KUKA KRL program: MyProgram_098().src

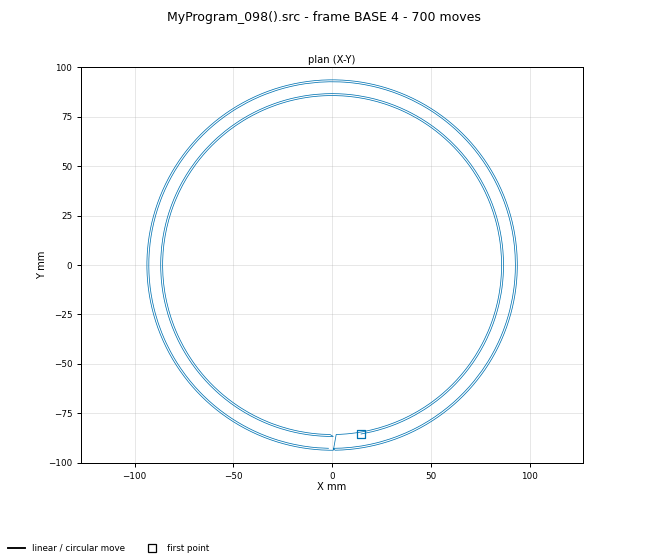
[picture p0: tool path of MyProgram_098().src in frame BASE 4, 700 of 700 moves have a stored position in this frame; points joined in program order, loops and branches not executed]
&ACCESS RVP
&REL 1
&PARAM TEMPLATE = C:\KRC\Roboter\Template\vorgabe
&PARAM EDITMASK = *
DEF MyProgram_098()
; ---- Setting reference (Base) ----
$BASE = BASE_DATA[4]

; --------------------------
; ---- Setting tool (TCP) ----
$TOOL = TOOL_DATA[3]
; --------------------------

$VEL.CP = VEL_APROX_PRINT
Startdeposition()
$VEL.CP = VEL_PRINT
LIN {X 14.6737,Y -85.5228,Z 90,A -84.3655,B 24.9258,C -1.989,E1 25.029,E2 169.2981} C_DIS
LIN {X 20.2856,Y -84.3677,Z 90,A -80.6832,B 24.9258,C -1.989,E1 25.0391,E2 165.6204} C_DIS
LIN {X 23.2527,Y -83.5992,Z 90,A -78.5972,B 24.9255,C -1.9933,E1 25.0447,E2 163.5279} C_DIS
LIN {X 26.6755,Y -82.5697,Z 90,A -75.7569,B 24.9241,C -2.0121,E1 25.0524,E2 160.6482} C_DIS
LIN {X 29.8401,Y -81.4795,Z 90,A -74.198,B 24.9255,C -1.9932,E1 25.0564,E2 159.1372} C_DIS
LIN {X 32.722,Y -80.3655,Z 90,A -72.0573,B 24.925,C -1.9994,E1 25.0619,E2 156.9867} C_DIS
LIN {X 35.8348,Y -79.0269,Z 90,A -69.6084,B 24.9243,C -2.0099,E1 25.0682,E2 154.5189} C_DIS
LIN {X 39.2577,Y -77.3837,Z 90,A -67.354,B 24.9246,C -2.0054,E1 25.0738,E2 152.2811} C_DIS
LIN {X 42.0598,Y -75.8972,Z 90,A -65.2291,B 24.9242,C -2.0101,E1 25.0791,E2 150.1513} C_DIS
LIN {X 46.6646,Y -73.1561,Z 90,A -62.0519,B 24.9247,C -2.0044,E1 25.0866,E2 146.9974} C_DIS
LIN {X 49.1042,Y -71.5429,Z 90,A -59.5239,B 24.9228,C -2.0285,E1 25.0926,E2 144.421} C_DIS
LIN {X 52.849,Y -68.8211,Z 90,A -56.8631,B 24.9234,C -2.0213,E1 25.0985,E2 141.7866} C_DIS
LIN {X 55.1312,Y -67.0079,Z 90,A -54.4863,B 24.9219,C -2.0411,E1 25.1037,E2 139.3722} C_DIS
LIN {X 57.7938,Y -64.7243,Z 90,A -52.5166,B 24.9224,C -2.0344,E1 25.1078,E2 137.426} C_DIS
LIN {X 60.5413,Y -62.1634,Z 90,A -50.2244,B 24.9224,C -2.0338,E1 25.1124,E2 135.1446} C_DIS
LIN {X 62.5386,Y -60.1521,Z 90,A -47.6066,B 24.9201,C -2.0643,E1 25.1176,E2 132.4661} C_DIS
LIN {X 64.9854,Y -57.5021,Z 90,A -45.8844,B 24.9214,C -2.0474,E1 25.1207,E2 130.7915} C_DIS
LIN {X 67.2469,Y -54.8385,Z 90,A -43.5543,B 24.9209,C -2.0542,E1 25.1249,E2 128.456} C_DIS
LIN {X 69.1339,Y -52.4405,Z 90,A -41.4737,B 24.9203,C -2.0619,E1 25.1285,E2 126.3672} C_DIS
LIN {X 71.5187,Y -49.139,Z 90,A -38.7198,B 24.9195,C -2.0715,E1 25.1329,E2 123.6039} C_DIS
LIN {X 73.5355,Y -46.0638,Z 90,A -35.8783,B 24.9179,C -2.0929,E1 25.1372,E2 120.7264} C_DIS
LIN {X 75.3159,Y -43.0915,Z 90,A -34.2647,B 24.9192,C -2.0758,E1 25.1394,E2 119.1613} C_DIS
LIN {X 76.7944,Y -40.3975,Z 90,A -32.1566,B 24.9185,C -2.0845,E1 25.1422,E2 117.0438} C_DIS
LIN {X 78.2764,Y -37.4454,Z 90,A -30.0963,B 24.9183,C -2.0868,E1 25.1447,E2 114.9892} C_DIS
LIN {X 80.2361,Y -33.0399,Z 90,A -26.7347,B 24.9171,C -2.1026,E1 25.1485,E2 111.6085} C_DIS
LIN {X 81.5916,Y -29.5328,Z 90,A -24.3204,B 24.9167,C -2.1079,E1 25.1508,E2 109.1953} C_DIS
LIN {X 82.6553,Y -26.4109,Z 90,A -22.0449,B 24.9159,C -2.1181,E1 25.1528,E2 106.9086} C_DIS
LIN {X 83.6832,Y -22.947,Z 90,A -19.8263,B 24.9157,C -2.1197,E1 25.1545,E2 104.6989} C_DIS
LIN {X 84.5153,Y -19.6601,Z 90,A -17.6432,B 24.9153,C -2.1248,E1 25.156,E2 102.5163} C_DIS
LIN {X 85.6245,Y -14.0659,Z 90,A -14.0298,B 24.9148,C -2.1314,E1 25.1579,E2 98.9085} C_DIS
LIN {X 86.0338,Y -11.2937,Z 90,A -12.3098,B 24.9147,C -2.1328,E1 25.1585,E2 97.1954} C_DIS
LIN {X 86.3255,Y -8.7923,Z 90,A -10.324,B 24.9133,C -2.1494,E1 25.1591,E2 95.182} C_DIS
LIN {X 86.6108,Y -5.3073,Z 90,A -7.9931,B 24.9127,C -2.1576,E1 25.1596,E2 92.8457} C_DIS
LIN {X 86.7486,Y -2.0565,Z 90,A -6.0028,B 24.9126,C -2.1589,E1 25.1598,E2 90.8641} C_DIS
LIN {X 86.7724,Y 0.3329,Z 90,A -4.3418,B 24.9119,C -2.1669,E1 25.1598,E2 89.1941} C_DIS
LIN {X 86.6858,Y 3.8646,Z 90,A -2.0074,B 24.9113,C -2.1744,E1 25.1595,E2 86.8558} C_DIS
LIN {X 86.4689,Y 7.2509,Z 90,A 0.1968,B 24.9108,C -2.1802,E1 25.1591,E2 84.651} C_DIS
LIN {X 86.1374,Y 10.4803,Z 90,A 2.3644,B 24.9102,C -2.1879,E1 25.1584,E2 82.4782} C_DIS
LIN {X 85.6296,Y 14.0351,Z 90,A 4.6778,B 24.9098,C -2.1933,E1 25.1574,E2 80.1656} C_DIS
LIN {X 85.1173,Y 16.8701,Z 90,A 6.6048,B 24.9092,C -2.2,E1 25.1564,E2 78.234} C_DIS
LIN {X 84.3903,Y 20.1931,Z 90,A 9.1136,B 24.9079,C -2.2161,E1 25.1548,E2 75.7017} C_DIS
LIN {X 83.2328,Y 24.5287,Z 90,A 11.6474,B 24.9084,C -2.2101,E1 25.1529,E2 73.1967} C_DIS
LIN {X 82.1608,Y 27.9101,Z 90,A 14.0041,B 24.9078,C -2.2176,E1 25.1509,E2 70.8357} C_DIS
LIN {X 81.0713,Y 30.9326,Z 90,A 16.1391,B 24.9072,C -2.2242,E1 25.1488,E2 68.6968} C_DIS
LIN {X 79.8847,Y 33.8794,Z 90,A 18.3025,B 24.9065,C -2.2326,E1 25.1465,E2 66.5256} C_DIS
LIN {X 78.4299,Y 37.1259,Z 90,A 20.3817,B 24.9067,C -2.2298,E1 25.1441,E2 64.4642} C_DIS
LIN {X 77.2493,Y 39.5206,Z 90,A 22.2334,B 24.9061,C -2.2378,E1 25.1417,E2 62.6036} C_DIS
LIN {X 75.2931,Y 43.1312,Z 90,A 24.6796,B 24.9062,C -2.236,E1 25.1385,E2 60.1744} C_DIS
LIN {X 74.1236,Y 45.1114,Z 90,A 26.4463,B 24.9052,C -2.2485,E1 25.1359,E2 58.3871} C_DIS
LIN {X 72.4967,Y 47.6821,Z 90,A 28.5137,B 24.9045,C -2.2557,E1 25.1328,E2 56.3132} C_DIS
LIN {X 70.2728,Y 50.9045,Z 90,A 31.1629,B 24.9038,C -2.2643,E1 25.1285,E2 53.6565} C_DIS
LIN {X 67.8225,Y 54.1259,Z 90,A 33.8258,B 24.9033,C -2.2704,E1 25.1239,E2 50.9918} C_DIS
LIN {X 65.5568,Y 56.8483,Z 90,A 36.1165,B 24.903,C -2.2742,E1 25.1198,E2 48.7027} C_DIS
LIN {X 63.2083,Y 59.4478,Z 90,A 38.8418,B 24.9013,C -2.2933,E1 25.1145,E2 45.9441} C_DIS
LIN {X 59.9076,Y 62.7742,Z 90,A 42.5078,B 24.8991,C -2.3192,E1 25.1071,E2 42.232} C_DIS
LIN {X 56.1883,Y 66.1228,Z 90,A 44.5817,B 24.9021,C -2.284,E1 25.1029,E2 40.2496} C_DIS
LIN {X 53.9722,Y 67.944,Z 90,A 46.6317,B 24.9014,C -2.2927,E1 25.0984,E2 38.1867} C_DIS
LIN {X 51.2627,Y 70.0105,Z 90,A 49.0796,B 24.9005,C -2.3032,E1 25.0929,E2 35.7226} C_DIS
LIN {X 48.4048,Y 72.0167,Z 90,A 51.2483,B 24.9005,C -2.3024,E1 25.0879,E2 33.5631} C_DIS
LIN {X 45.433,Y 73.9281,Z 90,A 53.5185,B 24.9005,C -2.3039,E1 25.0825,E2 31.2967} C_DIS
LIN {X 42.7507,Y 75.5114,Z 90,A 55.582,B 24.9001,C -2.3071,E1 25.0776,E2 29.232} C_DIS
LIN {X 40.0108,Y 76.9981,Z 90,A 57.4695,B 24.9004,C -2.3042,E1 25.0729,E2 27.3566} C_DIS
LIN {X 38.1158,Y 77.9535,Z 90,A 59.4503,B 24.8986,C -2.325,E1 25.0679,E2 25.3319} C_DIS
LIN {X 34.568,Y 79.5889,Z 90,A 61.647,B 24.8994,C -2.3153,E1 25.0623,E2 23.1635} C_DIS
LIN {X 31.3475,Y 80.9125,Z 90,A 63.8972,B 24.8994,C -2.316,E1 25.0565,E2 20.9168} C_DIS
LIN {X 28.2615,Y 82.0419,Z 90,A 66.0927,B 24.8991,C -2.3187,E1 25.0507,E2 18.7192} C_DIS
LIN {X 25.1389,Y 83.0518,Z 90,A 68.3337,B 24.8988,C -2.3228,E1 25.0447,E2 16.4727} C_DIS
LIN {X 21.4921,Y 84.0681,Z 90,A 70.6005,B 24.8993,C -2.3169,E1 25.0386,E2 14.2234} C_DIS
LIN {X 18.0347,Y 84.8782,Z 90,A 73.1039,B 24.8987,C -2.3231,E1 25.0318,E2 11.7086} C_DIS
LIN {X 12.9971,Y 85.7932,Z 90,A 76.2246,B 24.8994,C -2.316,E1 25.0233,E2 8.608} C_DIS
LIN {X 10.3284,Y 86.1552,Z 90,A 78.166,B 24.8989,C -2.3216,E1 25.0179,E2 6.655} C_DIS
LIN {X 7.047,Y 86.4852,Z 90,A 80.4053,B 24.8987,C -2.3237,E1 25.0116,E2 4.4119} C_DIS
LIN {X 3.4616,Y 86.7031,Z 90,A 82.8215,B 24.8986,C -2.325,E1 25.0049,E2 1.9934} C_DIS
LIN {X -0.1215,Y 86.7726,Z 90,A 85.1767,B 24.8986,C -2.3243,E1 24.9983,E2 -0.3598} C_DIS
LIN {X -3.486,Y 86.702,Z 90,A 88.3102,B 24.8962,C -2.3522,E1 24.9894,E2 -3.5602} C_DIS
LIN {X -8.2682,Y 86.3774,Z 90,A 90.3011,B 24.8995,C -2.3141,E1 24.9841,E2 -5.4615} C_DIS
LIN {X -10.9104,Y 86.0834,Z 90,A 92.2875,B 24.899,C -2.3202,E1 24.9785,E2 -7.4637} C_DIS
LIN {X -14.2435,Y 85.5948,Z 90,A 94.3609,B 24.8995,C -2.314,E1 24.9728,E2 -9.5243} C_DIS
LIN {X -18.3888,Y 84.8009,Z 90,A 97.2041,B 24.8995,C -2.3135,E1 24.9651,E2 -12.3694} C_DIS
LIN {X -20.776,Y 84.2481,Z 90,A 98.7974,B 24.8998,C -2.3112,E1 24.9607,E2 -13.9594} C_DIS
LIN {X -23.5949,Y 83.5022,Z 90,A 100.7155,B 24.9,C -2.309,E1 24.9556,E2 -15.8753} C_DIS
LIN {X -26.4229,Y 82.6514,Z 90,A 102.7582,B 24.9,C -2.3096,E1 24.9501,E2 -17.9229} C_DIS
LIN {X -29.1641,Y 81.7252,Z 90,A 104.6404,B 24.9002,C -2.3063,E1 24.9452,E2 -19.8011} C_DIS
LIN {X -32.9874,Y 80.2574,Z 90,A 106.9907,B 24.9014,C -2.2921,E1 24.9391,E2 -22.1227} C_DIS
LIN {X -36.8189,Y 78.5732,Z 90,A 110.1387,B 24.9008,C -2.2995,E1 24.931,E2 -25.2958} C_DIS
LIN {X -39.6003,Y 77.2086,Z 90,A 112.1958,B 24.901,C -2.2965,E1 24.9259,E2 -27.3513} C_DIS
LIN {X -42.1651,Y 75.8384,Z 90,A 114.2188,B 24.901,C -2.2963,E1 24.9209,E2 -29.3795} C_DIS
LIN {X -45.1483,Y 74.1011,Z 90,A 116.3655,B 24.9018,C -2.2883,E1 24.9158,E2 -31.5137} C_DIS
LIN {X -47.3167,Y 72.7365,Z 90,A 118.3871,B 24.9012,C -2.2948,E1 24.911,E2 -33.5573} C_DIS
LIN {X -51.1285,Y 70.1088,Z 90,A 121.2285,B 24.9023,C -2.2823,E1 24.9046,E2 -36.3788} C_DIS
LIN {X -54.2447,Y 67.7281,Z 90,A 123.6416,B 24.9032,C -2.2717,E1 24.8993,E2 -38.7753} C_DIS
LIN {X -58.0874,Y 64.4614,Z 90,A 126.9739,B 24.9038,C -2.2643,E1 24.8923,E2 -42.1029} C_DIS
LIN {X -60.725,Y 61.9821,Z 90,A 129.7326,B 24.9034,C -2.2693,E1 24.8866,E2 -44.8851} C_DIS
LIN {X -63.9027,Y 58.7008,Z 90,A 132.9799,B 24.9034,C -2.2686,E1 24.8804,E2 -48.1449} C_DIS
LIN {X -66.4847,Y 55.7609,Z 90,A 135.9724,B 24.903,C -2.2738,E1 24.875,E2 -51.1636} C_DIS
LIN {X -69.0469,Y 52.556,Z 90,A 137.9944,B 24.9053,C -2.2467,E1 24.8716,E2 -53.1304} C_DIS
LIN {X -71.9137,Y 48.5568,Z 90,A 141.2398,B 24.9061,C -2.2378,E1 24.8664,E2 -56.3704} C_DIS
LIN {X -73.8503,Y 45.5599,Z 90,A 143.623,B 24.9066,C -2.2319,E1 24.8629,E2 -58.7518} C_DIS
LIN {X -76.113,Y 41.6685,Z 90,A 146.4745,B 24.9076,C -2.2199,E1 24.8589,E2 -61.5896} C_DIS
LIN {X -77.4719,Y 39.0852,Z 90,A 148.5749,B 24.9076,C -2.2192,E1 24.8563,E2 -63.6994} C_DIS
LIN {X -78.9321,Y 36.0451,Z 90,A 150.8045,B 24.9082,C -2.2126,E1 24.8536,E2 -65.9255} C_DIS
LIN {X -80.0946,Y 33.3809,Z 90,A 152.5109,B 24.9091,C -2.2008,E1 24.8518,E2 -67.6132} C_DIS
LIN {X -81.3199,Y 30.2736,Z 90,A 155.3722,B 24.9082,C -2.2127,E1 24.8489,E2 -70.5189} C_DIS
LIN {X -82.6785,Y 26.3392,Z 90,A 157.478,B 24.9104,C -2.1859,E1 24.8471,E2 -72.5728} C_DIS
LIN {X -83.4112,Y 23.9161,Z 90,A 159.3644,B 24.9104,C -2.1868,E1 24.8456,E2 -74.4722} C_DIS
LIN {X -84.282,Y 20.6369,Z 90,A 161.5805,B 24.9109,C -2.179,E1 24.8441,E2 -76.6827} C_DIS
LIN {X -85.0114,Y 17.3897,Z 90,A 164.0725,B 24.9109,C -2.1804,E1 24.8426,E2 -79.1928} C_DIS
LIN {X -85.7162,Y 13.4951,Z 90,A 166.4556,B 24.912,C -2.1656,E1 24.8415,E2 -81.5545} C_DIS
LIN {X -86.3335,Y 8.7154,Z 90,A 169.3247,B 24.9136,C -2.1466,E1 24.8406,E2 -84.3954} C_DIS
LIN {X -86.6892,Y 3.7836,Z 90,A 172.8105,B 24.9139,C -2.1423,E1 24.8399,E2 -87.892} C_DIS
LIN {X -86.7687,Y 0.8198,Z 90,A 174.9512,B 24.914,C -2.1412,E1 24.8398,E2 -90.0429} C_DIS
LIN {X -86.7374,Y -2.451,Z 90,A 177.2545,B 24.9142,C -2.1384,E1 24.8399,E2 -92.3534} C_DIS
LIN {X -86.4654,Y -7.2952,Z 90,A -179.9825,B 24.916,C -2.1157,E1 24.8404,E2 -95.0789} C_DIS
LIN {X -86.0821,Y -10.921,Z 90,A -176.6927,B 24.9147,C -2.1332,E1 24.8415,E2 -98.4302} C_DIS
LIN {X -85.5867,Y -14.2915,Z 90,A -174.745,B 24.9159,C -2.1176,E1 24.8424,E2 -100.3521} C_DIS
LIN {X -85.039,Y -17.2554,Z 90,A -172.9537,B 24.9168,C -2.1057,E1 24.8433,E2 -102.1257} C_DIS
LIN {X -84.2536,Y -20.7533,Z 90,A -170.363,B 24.9169,C -2.1049,E1 24.845,E2 -104.7296} C_DIS
LIN {X -83.1494,Y -24.8099,Z 90,A -167.7527,B 24.9179,C -2.0918,E1 24.847,E2 -107.3236} C_DIS
LIN {X -82.053,Y -28.2298,Z 90,A -165.3254,B 24.9184,C -2.0863,E1 24.8491,E2 -109.7518} C_DIS
LIN {X -80.8131,Y -31.6004,Z 90,A -163.0692,B 24.9192,C -2.0761,E1 24.8514,E2 -111.9964} C_DIS
LIN {X -79.3475,Y -35.1214,Z 90,A -160.6221,B 24.9199,C -2.0669,E1 24.854,E2 -114.435} C_DIS
LIN {X -78.0432,Y -37.9308,Z 90,A -158.562,B 24.9203,C -2.0616,E1 24.8565,E2 -116.4936} C_DIS
LIN {X -76.8182,Y -40.3523,Z 90,A -156.889,B 24.9209,C -2.0533,E1 24.8586,E2 -118.1557} C_DIS
LIN {X -75.5782,Y -42.6311,Z 90,A -154.8456,B 24.9206,C -2.0582,E1 24.8614,E2 -120.2216} C_DIS
LIN {X -73.7903,Y -45.6559,Z 90,A -152.6186,B 24.9212,C -2.0494,E1 24.8646,E2 -122.4392} C_DIS
LIN {X -72.1751,Y -48.1698,Z 90,A -150.5085,B 24.9213,C -2.0483,E1 24.8679,E2 -124.5573} C_DIS
LIN {X -70.7147,Y -50.287,Z 90,A -148.9125,B 24.9219,C -2.0411,E1 24.8704,E2 -126.144} C_DIS
LIN {X -68.7632,Y -52.9241,Z 90,A -146.7243,B 24.9222,C -2.0365,E1 24.8741,E2 -128.3317} C_DIS
LIN {X -66.659,Y -55.5512,Z 90,A -144.4803,B 24.9226,C -2.032,E1 24.8781,E2 -130.5752} C_DIS
LIN {X -63.9474,Y -58.652,Z 90,A -141.8407,B 24.9232,C -2.0235,E1 24.8829,E2 -133.2065} C_DIS
LIN {X -61.8709,Y -60.8388,Z 90,A -139.7469,B 24.9233,C -2.0223,E1 24.887,E2 -135.3064} C_DIS
LIN {X -58.6643,Y -63.9362,Z 90,A -137.0467,B 24.9243,C -2.009,E1 24.8924,E2 -137.9862} C_DIS
LIN {X -56.837,Y -65.5667,Z 90,A -135.1434,B 24.9239,C -2.0144,E1 24.8965,E2 -139.9097} C_DIS
LIN {X -54.3681,Y -67.6282,Z 90,A -133.0279,B 24.9242,C -2.0102,E1 24.901,E2 -142.0232} C_DIS
LIN {X -51.5777,Y -69.7799,Z 90,A -130.6538,B 24.9244,C -2.0076,E1 24.9063,E2 -144.3996} C_DIS
LIN {X -48.8844,Y -71.6919,Z 90,A -128.8231,B 24.9255,C -1.9935,E1 24.9105,E2 -146.203} C_DIS
LIN {X -46.8547,Y -73.034,Z 90,A -126.9337,B 24.925,C -1.9995,E1 24.9149,E2 -148.1129} C_DIS
LIN {X -44.0516,Y -74.7583,Z 90,A -124.7119,B 24.9252,C -1.9978,E1 24.9202,E2 -150.3375} C_DIS
LIN {X -41.0669,Y -76.4393,Z 90,A -121.962,B 24.9243,C -2.0097,E1 24.9271,E2 -153.1235} C_DIS
LIN {X -37.487,Y -78.2564,Z 90,A -119.7057,B 24.9254,C -1.9944,E1 24.9327,E2 -155.3492} C_DIS
LIN {X -34.2603,Y -79.7228,Z 90,A -117.4046,B 24.9257,C -1.9906,E1 24.9385,E2 -157.6469} C_DIS
LIN {X -31.2553,Y -80.9487,Z 90,A -115.2188,B 24.9257,C -1.9898,E1 24.9442,E2 -159.8356} C_DIS
LIN {X -28.152,Y -82.0793,Z 90,A -113.0731,B 24.926,C -1.9869,E1 24.9499,E2 -161.9786} C_DIS
LIN {X -25.6504,Y -82.8939,Z 90,A -111.4199,B 24.9263,C -1.983,E1 24.9542,E2 -163.6255} C_DIS
LIN {X -21.7868,Y -83.9923,Z 90,A -108.778,B 24.9264,C -1.981,E1 24.9613,E2 -166.2667} C_DIS
LIN {X -18.6922,Y -84.7348,Z 90,A -106.5901,B 24.9263,C -1.9827,E1 24.9673,E2 -168.4615} C_DIS
LIN {X -16.0435,Y -85.2765,Z 90,A -104.7441,B 24.9263,C -1.9839,E1 24.9724,E2 -170.3124} C_DIS
LIN {X -12.5033,Y -85.8667,Z 90,A -102.4021,B 24.9263,C -1.9824,E1 24.9789,E2 -172.6529} C_DIS
LIN {X -9.1954,Y -86.2833,Z 90,A -100.2446,B 24.9264,C -1.9807,E1 24.9848,E2 -174.8078} C_DIS
LIN {X -5.6527,Y -86.5877,Z 90,A -97.8304,B 24.9263,C -1.9828,E1 24.9916,E2 -177.2279} C_DIS
LIN {X -2.1762,Y -86.7458,Z 90,A -95.5345,B 24.9263,C -1.983,E1 24.998,E2 -179.5247} C_DIS
LIN {X 0.5801,Y -86.7688,Z 90,A -94.5554,B 24.9282,C -1.9566,E1 25.0005,E2 -180.441} C_DIS
Enddeposition()
LIN {X 0.5801,Y -86.7688,Z 90,A -94.5554,B 24.9282,C -1.9566,E1 25.0005,E2 -180.441} C_DIS
Startdeposition()
$VEL.CP = VEL_PRINT
LIN {X -1.0607,Y -85.7862,Z 90,A -95.749,B 24.9272,C -1.9704,E1 24.9973,E2 -179.2802} C_DIS
LIN {X -3.1996,Y -85.7329,Z 90,A -97.1333,B 24.9272,C -1.9716,E1 24.9934,E2 -177.8985} C_DIS
LIN {X -5.3003,Y -85.6287,Z 90,A -98.5378,B 24.9272,C -1.9716,E1 24.9895,E2 -176.4935} C_DIS
LIN {X -7.3979,Y -85.4731,Z 90,A -99.9428,B 24.9272,C -1.9716,E1 24.9856,E2 -175.0879} C_DIS
LIN {X -10.0614,Y -85.1992,Z 90,A -101.8399,B 24.9274,C -1.9684,E1 24.9803,E2 -173.1822} C_DIS
LIN {X -12.629,Y -84.858,Z 90,A -103.4847,B 24.9271,C -1.9714,E1 24.9758,E2 -171.5432} C_DIS
LIN {X -14.6696,Y -84.5294,Z 90,A -104.8659,B 24.9271,C -1.9718,E1 24.972,E2 -170.1616} C_DIS
LIN {X -16.773,Y -84.137,Z 90,A -106.2741,B 24.9271,C -1.9729,E1 24.9681,E2 -168.7546} C_DIS
LIN {X -18.795,Y -83.7088,Z 90,A -107.9321,B 24.9276,C -1.9651,E1 24.9635,E2 -167.076} C_DIS
LIN {X -21.9151,Y -82.9463,Z 90,A -109.8016,B 24.9269,C -1.9747,E1 24.9585,E2 -165.2266} C_DIS
LIN {X -23.9017,Y -82.3961,Z 90,A -111.2246,B 24.9269,C -1.9742,E1 24.9547,E2 -163.8} C_DIS
LIN {X -25.9433,Y -81.7761,Z 90,A -112.637,B 24.9269,C -1.9756,E1 24.9509,E2 -162.3886} C_DIS
LIN {X -27.914,Y -81.1247,Z 90,A -114.0199,B 24.9267,C -1.9768,E1 24.9473,E2 -161.006} C_DIS
LIN {X -29.9274,Y -80.4035,Z 90,A -115.451,B 24.9267,C -1.978,E1 24.9435,E2 -159.5747} C_DIS
LIN {X -31.8885,Y -79.6461,Z 90,A -116.8376,B 24.9265,C -1.9798,E1 24.9399,E2 -158.1896} C_DIS
LIN {X -34.058,Y -78.7416,Z 90,A -118.2913,B 24.9261,C -1.985,E1 24.9362,E2 -156.7447} C_DIS
LIN {X -35.7637,Y -77.9829,Z 90,A -119.7008,B 24.9264,C -1.9815,E1 24.9326,E2 -155.3235} C_DIS
LIN {X -37.6857,Y -77.0723,Z 90,A -121.0789,B 24.9262,C -1.9844,E1 24.9291,E2 -153.9488} C_DIS
LIN {X -39.5187,Y -76.149,Z 90,A -122.6453,B 24.9265,C -1.9803,E1 24.9252,E2 -152.3684} C_DIS
LIN {X -42.2912,Y -74.6449,Z 90,A -124.593,B 24.9259,C -1.9878,E1 24.9205,E2 -150.4331} C_DIS
LIN {X -44.1074,Y -73.5863,Z 90,A -126.0232,B 24.9259,C -1.9891,E1 24.917,E2 -149.0014} C_DIS
LIN {X -45.8971,Y -72.4835,Z 90,A -127.4109,B 24.9256,C -1.9916,E1 24.9137,E2 -147.6155} C_DIS
LIN {X -47.6592,Y -71.3373,Z 90,A -129.0095,B 24.9259,C -1.9882,E1 24.91,E2 -146.0033} C_DIS
LIN {X -50.2582,Y -69.5307,Z 90,A -130.9487,B 24.9252,C -1.9968,E1 24.9056,E2 -144.078} C_DIS
LIN {X -52.3715,Y -67.9511,Z 90,A -132.8208,B 24.9252,C -1.9967,E1 24.9014,E2 -142.1989} C_DIS
LIN {X -54.8478,Y -65.9686,Z 90,A -134.9408,B 24.925,C -2.0005,E1 24.8968,E2 -140.0801} C_DIS
LIN {X -57.2356,Y -63.9079,Z 90,A -137.0745,B 24.9247,C -2.0038,E1 24.8923,E2 -137.9459} C_DIS
LIN {X -59.555,Y -61.7522,Z 90,A -139.1913,B 24.9244,C -2.0081,E1 24.8881,E2 -135.8304} C_DIS
LIN {X -61.783,Y -59.523,Z 90,A -141.304,B 24.9241,C -2.0123,E1 24.8839,E2 -133.7188} C_DIS
LIN {X -63.9035,Y -57.2406,Z 90,A -143.414,B 24.9238,C -2.0161,E1 24.8799,E2 -131.6085} C_DIS
LIN {X -65.995,Y -54.816,Z 90,A -145.5359,B 24.9234,C -2.0214,E1 24.8761,E2 -129.4897} C_DIS
LIN {X -67.9545,Y -52.3672,Z 90,A -147.6485,B 24.923,C -2.0259,E1 24.8725,E2 -127.3778} C_DIS
LIN {X -69.5484,Y -50.2334,Z 90,A -149.3087,B 24.9225,C -2.0336,E1 24.8697,E2 -125.7278} C_DIS
LIN {X -70.7582,Y -48.5146,Z 90,A -150.7527,B 24.9223,C -2.036,E1 24.8674,E2 -124.2823} C_DIS
LIN {X -72.0134,Y -46.6296,Z 90,A -152.1489,B 24.9217,C -2.0431,E1 24.8653,E2 -122.8962} C_DIS
LIN {X -73.0617,Y -44.9707,Z 90,A -153.5769,B 24.9217,C -2.0431,E1 24.8632,E2 -121.4611} C_DIS
LIN {X -74.1419,Y -43.1665,Z 90,A -154.9895,B 24.9215,C -2.0466,E1 24.8612,E2 -120.0495} C_DIS
LIN {X -75.1603,Y -41.3683,Z 90,A -156.5048,B 24.9215,C -2.0466,E1 24.8591,E2 -118.526} C_DIS
LIN {X -76.1728,Y -39.4724,Z 90,A -157.7983,B 24.9209,C -2.0544,E1 24.8574,E2 -117.2444} C_DIS
LIN {X -77.1159,Y -37.5966,Z 90,A -159.2105,B 24.9206,C -2.058,E1 24.8557,E2 -115.8333} C_DIS
LIN {X -77.9979,Y -35.7314,Z 90,A -160.6374,B 24.9204,C -2.0605,E1 24.854,E2 -114.4044} C_DIS
LIN {X -78.9641,Y -33.5389,Z 90,A -162.3566,B 24.9203,C -2.0618,E1 24.8521,E2 -112.6788} C_DIS
LIN {X -80.0453,Y -30.8731,Z 90,A -164.1838,B 24.9197,C -2.0699,E1 24.8502,E2 -110.8609} C_DIS
LIN {X -80.7902,Y -28.8673,Z 90,A -165.5791,B 24.9193,C -2.0751,E1 24.8489,E2 -109.4698} C_DIS
LIN {X -81.4736,Y -26.8782,Z 90,A -166.9947,B 24.919,C -2.0789,E1 24.8476,E2 -108.0554} C_DIS
LIN {X -82.1332,Y -24.7879,Z 90,A -168.4399,B 24.9186,C -2.0838,E1 24.8464,E2 -106.6135} C_DIS
LIN {X -82.6898,Y -22.8648,Z 90,A -169.8337,B 24.9184,C -2.0863,E1 24.8454,E2 -105.2175} C_DIS
LIN {X -83.2328,Y -20.8004,Z 90,A -171.2694,B 24.9181,C -2.0903,E1 24.8444,E2 -103.7831} C_DIS
LIN {X -83.7168,Y -18.758,Z 90,A -172.8066,B 24.9181,C -2.0909,E1 24.8434,E2 -102.2383} C_DIS
LIN {X -84.2766,Y -16.0506,Z 90,A -174.6165,B 24.9175,C -2.0976,E1 24.8424,E2 -100.4337} C_DIS
LIN {X -84.7074,Y -13.6027,Z 90,A -176.2316,B 24.917,C -2.104,E1 24.8417,E2 -98.8242} C_DIS
LIN {X -85.019,Y -11.4944,Z 90,A -177.6213,B 24.9166,C -2.1094,E1 24.8411,E2 -97.4391} C_DIS
LIN {X -85.2746,Y -9.4136,Z 90,A -179.0314,B 24.9162,C -2.1135,E1 24.8407,E2 -96.0304} C_DIS
LIN {X -85.4792,Y -7.3267,Z 90,A 179.5357,B 24.9159,C -2.117,E1 24.8403,E2 -94.5974} C_DIS
LIN {X -85.6348,Y -5.1998,Z 90,A 178.1237,B 24.9156,C -2.1219,E1 24.84,E2 -93.1885} C_DIS
LIN {X -85.7352,Y -3.1414,Z 90,A 176.6932,B 24.9153,C -2.1248,E1 24.8399,E2 -91.7562} C_DIS
LIN {X -85.7872,Y -0.9416,Z 90,A 175.3696,B 24.9146,C -2.1335,E1 24.8398,E2 -90.4455} C_DIS
LIN {X -85.7659,Y 2.141,Z 90,A 173.161,B 24.9144,C -2.1359,E1 24.8398,E2 -88.2294} C_DIS
LIN {X -85.6866,Y 4.262,Z 90,A 171.7353,B 24.9141,C -2.1403,E1 24.84,E2 -86.8054} C_DIS
LIN {X -85.5599,Y 6.3171,Z 90,A 170.3269,B 24.9138,C -2.1437,E1 24.8403,E2 -85.3969} C_DIS
LIN {X -85.3739,Y 8.4644,Z 90,A 168.8986,B 24.9134,C -2.1487,E1 24.8407,E2 -83.9717} C_DIS
LIN {X -85.146,Y 10.5142,Z 90,A 167.5121,B 24.9131,C -2.1528,E1 24.8411,E2 -82.5868} C_DIS
LIN {X -84.8252,Y 12.841,Z 90,A 166.0606,B 24.9124,C -2.161,E1 24.8417,E2 -81.1463} C_DIS
LIN {X -84.5303,Y 14.6644,Z 90,A 164.6874,B 24.9124,C -2.1611,E1 24.8423,E2 -79.7652} C_DIS
LIN {X -84.1352,Y 16.782,Z 90,A 163.2624,B 24.912,C -2.1661,E1 24.8431,E2 -78.3435} C_DIS
LIN {X -83.7069,Y 18.803,Z 90,A 161.8501,B 24.9117,C -2.1695,E1 24.8439,E2 -76.9312} C_DIS
LIN {X -83.212,Y 20.8838,Z 90,A 160.4117,B 24.9114,C -2.1738,E1 24.8449,E2 -75.4945} C_DIS
LIN {X -82.6844,Y 22.8843,Z 90,A 159.021,B 24.911,C -2.1778,E1 24.8459,E2 -74.1055} C_DIS
LIN {X -82.0889,Y 24.9358,Z 90,A 157.6033,B 24.9107,C -2.1825,E1 24.847,E2 -72.6907} C_DIS
LIN {X -81.4626,Y 26.9121,Z 90,A 155.9315,B 24.9109,C -2.179,E1 24.8484,E2 -71.0009} C_DIS
LIN {X -80.3714,Y 30.0121,Z 90,A 153.8101,B 24.9102,C -2.1877,E1 24.8505,E2 -68.8884} C_DIS
LIN {X -79.2584,Y 32.8406,Z 90,A 151.9358,B 24.9094,C -2.1982,E1 24.8524,E2 -67.0285} C_DIS
LIN {X -78.415,Y 34.806,Z 90,A 150.4978,B 24.909,C -2.2022,E1 24.854,E2 -65.5922} C_DIS
LIN {X -77.5543,Y 36.6844,Z 90,A 149.0866,B 24.9088,C -2.2054,E1 24.8557,E2 -64.1811} C_DIS
LIN {X -76.632,Y 38.5739,Z 90,A 147.6946,B 24.9084,C -2.2099,E1 24.8574,E2 -62.7923} C_DIS
LIN {X -75.6318,Y 40.4991,Z 90,A 146.2609,B 24.908,C -2.2146,E1 24.8592,E2 -61.362} C_DIS
LIN {X -74.6376,Y 42.304,Z 90,A 144.8532,B 24.9077,C -2.2177,E1 24.8612,E2 -59.9543} C_DIS
LIN {X -73.5807,Y 44.1167,Z 90,A 143.3428,B 24.9077,C -2.2186,E1 24.8633,E2 -58.4384} C_DIS
LIN {X -72.4793,Y 45.9037,Z 90,A 142.0318,B 24.9071,C -2.2251,E1 24.8652,E2 -57.1361} C_DIS
LIN {X -71.3344,Y 47.6635,Z 90,A 140.5247,B 24.9071,C -2.2261,E1 24.8676,E2 -55.6239} C_DIS
LIN {X -70.0838,Y 49.4831,Z 90,A 139.1293,B 24.9065,C -2.2323,E1 24.8698,E2 -54.2365} C_DIS
LIN {X -68.8742,Y 51.1536,Z 90,A 137.5497,B 24.9067,C -2.2304,E1 24.8724,E2 -52.6447} C_DIS
LIN {X -66.967,Y 53.6266,Z 90,A 135.4361,B 24.9063,C -2.2351,E1 24.8761,E2 -50.5324} C_DIS
LIN {X -64.9645,Y 56.0359,Z 90,A 133.4017,B 24.9057,C -2.2421,E1 24.8797,E2 -48.5053} C_DIS
LIN {X -63.1238,Y 58.0994,Z 90,A 131.5741,B 24.9053,C -2.2473,E1 24.8831,E2 -46.6819} C_DIS
LIN {X -61.0028,Y 60.3224,Z 90,A 129.5142,B 24.9049,C -2.252,E1 24.8871,E2 -44.6245} C_DIS
LIN {X -58.7656,Y 62.5039,Z 90,A 127.4236,B 24.9044,C -2.2568,E1 24.8914,E2 -42.5368} C_DIS
LIN {X -56.3922,Y 64.6534,Z 90,A 125.2696,B 24.9041,C -2.2613,E1 24.8958,E2 -40.3847} C_DIS
LIN {X -53.9879,Y 66.6742,Z 90,A 123.1557,B 24.9037,C -2.2654,E1 24.9004,E2 -38.2726} C_DIS
LIN {X -51.9095,Y 68.3064,Z 90,A 121.524,B 24.9031,C -2.2729,E1 24.904,E2 -36.6527} C_DIS
LIN {X -50.1425,Y 69.6133,Z 90,A 120.1123,B 24.9027,C -2.2775,E1 24.9071,E2 -35.2471} C_DIS
LIN {X -48.5097,Y 70.7615,Z 90,A 118.6733,B 24.9027,C -2.2771,E1 24.9104,E2 -33.8022} C_DIS
LIN {X -46.7436,Y 71.9403,Z 90,A 117.2848,B 24.9024,C -2.2807,E1 24.9137,E2 -32.4177} C_DIS
LIN {X -44.9676,Y 73.0635,Z 90,A 115.8529,B 24.9023,C -2.2825,E1 24.9171,E2 -30.9856} C_DIS
LIN {X -43.1644,Y 74.1431,Z 90,A 114.285,B 24.9025,C -2.2803,E1 24.9209,E2 -29.4077} C_DIS
LIN {X -40.4433,Y 75.6621,Z 90,A 112.3329,B 24.9018,C -2.2875,E1 24.9256,E2 -27.4673} C_DIS
LIN {X -38.5776,Y 76.6301,Z 90,A 110.9265,B 24.9016,C -2.2897,E1 24.9291,E2 -26.0623} C_DIS
LIN {X -36.6889,Y 77.5521,Z 90,A 109.3956,B 24.9018,C -2.2882,E1 24.933,E2 -24.5239} C_DIS
LIN {X -34.7313,Y 78.4481,Z 90,A 107.8724,B 24.9018,C -2.2879,E1 24.9369,E2 -22.9963} C_DIS
LIN {X -31.8389,Y 79.666,Z 90,A 105.9897,B 24.901,C -2.297,E1 24.9417,E2 -21.131} C_DIS
LIN {X -29.8454,Y 80.4339,Z 90,A 104.5615,B 24.9009,C -2.2988,E1 24.9454,E2 -19.7041} C_DIS
LIN {X -27.9016,Y 81.1289,Z 90,A 103.1572,B 24.9008,C -2.2998,E1 24.9491,E2 -18.2994} C_DIS
LIN {X -25.9066,Y 81.7879,Z 90,A 101.6069,B 24.901,C -2.2971,E1 24.9533,E2 -16.7399} C_DIS
LIN {X -22.8852,Y 82.6842,Z 90,A 99.6609,B 24.9004,C -2.304,E1 24.9584,E2 -14.8073} C_DIS
LIN {X -20.8185,Y 83.2284,Z 90,A 98.2319,B 24.9003,C -2.3054,E1 24.9623,E2 -13.3793} C_DIS
LIN {X -18.1891,Y 83.8409,Z 90,A 96.2703,B 24.9005,C -2.3023,E1 24.9677,E2 -11.408} C_DIS
LIN {X -15.3015,Y 84.4157,Z 90,A 94.2969,B 24.9005,C -2.3037,E1 24.9731,E2 -9.4357} C_DIS
LIN {X -12.546,Y 84.8703,Z 90,A 92.5864,B 24.8999,C -2.3095,E1 24.9778,E2 -7.7376} C_DIS
LIN {X -10.4979,Y 85.1481,Z 90,A 91.0453,B 24.9003,C -2.3056,E1 24.9821,E2 -6.1859} C_DIS
LIN {X -6.9567,Y 85.5088,Z 90,A 88.6164,B 24.9003,C -2.3052,E1 24.9888,E2 -3.7549} C_DIS
LIN {X -4.1566,Y 85.6918,Z 90,A 86.8398,B 24.9,C -2.3088,E1 24.9938,E2 -1.9863} C_DIS
LIN {X -1.5014,Y 85.7781,Z 90,A 85.0859,B 24.8999,C -2.3099,E1 24.9986,E2 -0.2349} C_DIS
LIN {X 1.0568,Y 85.7863,Z 90,A 83.4421,B 24.8997,C -2.3122,E1 25.0032,E2 1.4035} C_DIS
LIN {X 3.1958,Y 85.7331,Z 90,A 82.0573,B 24.8996,C -2.3137,E1 25.0071,E2 2.7845} C_DIS
LIN {X 5.2965,Y 85.629,Z 90,A 80.6515,B 24.8996,C -2.3137,E1 25.011,E2 4.1897} C_DIS
LIN {X 8.4156,Y 85.3791,Z 90,A 78.5189,B 24.8996,C -2.3122,E1 25.0169,E2 6.3247} C_DIS
LIN {X 10.506,Y 85.1471,Z 90,A 77.1364,B 24.8996,C -2.3126,E1 25.0208,E2 7.7052} C_DIS
LIN {X 12.626,Y 84.8584,Z 90,A 75.4036,B 24.9005,C -2.3029,E1 25.0256,E2 9.4595} C_DIS
LIN {X 16.4118,Y 84.207,Z 90,A 73.0838,B 24.8999,C -2.3095,E1 25.0319,E2 11.761} C_DIS
LIN {X 18.8114,Y 83.705,Z 90,A 71.5107,B 24.8999,C -2.3107,E1 25.0362,E2 13.3292} C_DIS
LIN {X 20.8878,Y 83.211,Z 90,A 70.0869,B 24.8999,C -2.3099,E1 25.0401,E2 14.7527} C_DIS
LIN {X 22.9193,Y 82.6745,Z 90,A 68.7029,B 24.8999,C -2.3096,E1 25.0438,E2 16.1352} C_DIS
LIN {X 24.9442,Y 82.0863,Z 90,A 67.3008,B 24.8999,C -2.3088,E1 25.0476,E2 17.5369} C_DIS
LIN {X 26.948,Y 81.4505,Z 90,A 65.8994,B 24.9001,C -2.3078,E1 25.0513,E2 18.9381} C_DIS
LIN {X 28.9014,Y 80.7782,Z 90,A 64.4789,B 24.9003,C -2.3053,E1 25.055,E2 20.3617} C_DIS
LIN {X 30.989,Y 79.9999,Z 90,A 63.0618,B 24.9003,C -2.3061,E1 25.0587,E2 21.7738} C_DIS
LIN {X 32.8356,Y 79.2605,Z 90,A 61.6344,B 24.9006,C -2.3016,E1 25.0624,E2 23.2086} C_DIS
LIN {X 34.8509,Y 78.3947,Z 90,A 60.2401,B 24.9006,C -2.3022,E1 25.066,E2 24.5979} C_DIS
LIN {X 37.1245,Y 77.3428,Z 90,A 58.4331,B 24.9011,C -2.296,E1 25.0706,E2 26.415} C_DIS
LIN {X 39.5161,Y 76.1504,Z 90,A 56.7582,B 24.901,C -2.2972,E1 25.0747,E2 28.0825} C_DIS
LIN {X 41.3695,Y 75.1597,Z 90,A 55.3805,B 24.901,C -2.2962,E1 25.0781,E2 29.4587} C_DIS
LIN {X 43.1981,Y 74.1238,Z 90,A 53.9802,B 24.9012,C -2.2943,E1 25.0815,E2 30.8593} C_DIS
LIN {X 45.5647,Y 72.6912,Z 90,A 52.0703,B 24.9017,C -2.2895,E1 25.0861,E2 32.7745} C_DIS
LIN {X 48.1253,Y 71.0217,Z 90,A 49.997,B 24.902,C -2.2852,E1 25.0909,E2 34.8511} C_DIS
LIN {X 50.2972,Y 69.5022,Z 90,A 48.3646,B 24.902,C -2.2867,E1 25.0946,E2 36.4744} C_DIS
LIN {X 52.3695,Y 67.9527,Z 90,A 46.5105,B 24.9025,C -2.2795,E1 25.0987,E2 38.3386} C_DIS
LIN {X 54.8448,Y 65.9711,Z 90,A 44.3896,B 24.9029,C -2.2755,E1 25.1033,E2 40.461} C_DIS
LIN {X 57.2492,Y 63.8957,Z 90,A 42.2844,B 24.9032,C -2.2719,E1 25.1078,E2 42.5665} C_DIS
LIN {X 59.552,Y 61.7551,Z 90,A 40.1983,B 24.9035,C -2.268,E1 25.112,E2 44.6531} C_DIS
LIN {X 61.7893,Y 59.5166,Z 90,A 38.0898,B 24.9039,C -2.2636,E1 25.1161,E2 46.7629} C_DIS
LIN {X 63.9339,Y 57.2065,Z 90,A 35.9969,B 24.9042,C -2.2594,E1 25.1201,E2 48.8566} C_DIS
LIN {X 65.9925,Y 54.819,Z 90,A 33.9115,B 24.9046,C -2.2552,E1 25.1238,E2 50.9425} C_DIS
LIN {X 68.0374,Y 52.2596,Z 90,A 31.7709,B 24.9049,C -2.2515,E1 25.1275,E2 53.0817} C_DIS
LIN {X 69.5527,Y 50.2275,Z 90,A 29.9504,B 24.9056,C -2.2431,E1 25.1305,E2 54.9133} C_DIS
LIN {X 71.3594,Y 47.6256,Z 90,A 28.051,B 24.9055,C -2.2449,E1 25.1335,E2 56.799} C_DIS
LIN {X 72.4852,Y 45.8945,Z 90,A 26.658,B 24.9058,C -2.2409,E1 25.1356,E2 58.1945} C_DIS
LIN {X 73.6061,Y 44.0741,Z 90,A 25.0731,B 24.9066,C -2.2319,E1 25.1379,E2 59.7926} C_DIS
LIN {X 75.1912,Y 41.3114,Z 90,A 23.1417,B 24.9065,C -2.2327,E1 25.1406,E2 61.712} C_DIS
LIN {X 76.4302,Y 38.9688,Z 90,A 21.2829,B 24.9071,C -2.2249,E1 25.143,E2 63.5794} C_DIS
LIN {X 77.5557,Y 36.6813,Z 90,A 19.4784,B 24.9078,C -2.2167,E1 25.1452,E2 65.3937} C_DIS
LIN {X 78.8705,Y 33.761,Z 90,A 17.4116,B 24.9081,C -2.2131,E1 25.1475,E2 67.4578} C_DIS
LIN {X 80.0449,Y 30.8743,Z 90,A 15.4781,B 24.9082,C -2.212,E1 25.1495,E2 69.383} C_DIS
LIN {X 80.7893,Y 28.8697,Z 90,A 14.0314,B 24.9086,C -2.2072,E1 25.1509,E2 70.833} C_DIS
LIN {X 81.4769,Y 26.8677,Z 90,A 12.7006,B 24.9087,C -2.2058,E1 25.152,E2 72.1596} C_DIS
LIN {X 82.1665,Y 24.6755,Z 90,A 11.2726,B 24.9088,C -2.2049,E1 25.1532,E2 73.5817} C_DIS
LIN {X 82.6832,Y 22.8888,Z 90,A 9.917,B 24.9094,C -2.1972,E1 25.1543,E2 74.9475} C_DIS
LIN {X 83.2264,Y 20.8267,Z 90,A 8.2598,B 24.9105,C -2.185,E1 25.1554,E2 76.6241} C_DIS
LIN {X 83.9332,Y 17.7659,Z 90,A 6.3974,B 24.9103,C -2.1865,E1 25.1565,E2 78.4721} C_DIS
LIN {X 84.3499,Y 15.6672,Z 90,A 5.022,B 24.9105,C -2.1839,E1 25.1573,E2 79.8456} C_DIS
LIN {X 84.7031,Y 13.6307,Z 90,A 3.6083,B 24.911,C -2.1785,E1 25.1579,E2 81.2638} C_DIS
LIN {X 85.0165,Y 11.5141,Z 90,A 1.9769,B 24.9119,C -2.1671,E1 25.1586,E2 82.9125} C_DIS
LIN {X 85.3799,Y 8.4069,Z 90,A 0.1133,B 24.9119,C -2.1682,E1 25.1591,E2 84.7625} C_DIS
LIN {X 85.5604,Y 6.3113,Z 90,A -1.2818,B 24.9122,C -2.164,E1 25.1594,E2 86.1591} C_DIS
LIN {X 85.6894,Y 4.212,Z 90,A -2.6556,B 24.9124,C -2.1606,E1 25.1596,E2 87.5327} C_DIS
LIN {X 85.7676,Y 2.0738,Z 90,A -4.1021,B 24.9129,C -2.1555,E1 25.1598,E2 88.9828} C_DIS
LIN {X 85.7915,Y -0.388,Z 90,A -5.917,B 24.9138,C -2.1444,E1 25.1598,E2 90.8132} C_DIS
LIN {X 85.733,Y -3.1965,Z 90,A -7.5468,B 24.9136,C -2.1468,E1 25.1596,E2 92.4276} C_DIS
LIN {X 85.629,Y -5.2969,Z 90,A -9.1443,B 24.9145,C -2.1356,E1 25.1594,E2 94.0418} C_DIS
LIN {X 85.3801,Y -8.4049,Z 90,A -11.0505,B 24.9145,C -2.135,E1 25.1589,E2 95.9383} C_DIS
LIN {X 85.1485,Y -10.4949,Z 90,A -12.5795,B 24.9152,C -2.1262,E1 25.1584,E2 97.4789} C_DIS
LIN {X 84.7292,Y -13.4617,Z 90,A -14.4492,B 24.9154,C -2.1243,E1 25.1576,E2 99.3421} C_DIS
LIN {X 84.3379,Y -15.7322,Z 90,A -16.1184,B 24.9161,C -2.1149,E1 25.1568,E2 101.0236} C_DIS
LIN {X 83.705,Y -18.8114,Z 90,A -18.0242,B 24.9161,C -2.1149,E1 25.1557,E2 102.9185} C_DIS
LIN {X 83.2111,Y -20.8872,Z 90,A -19.4394,B 24.9164,C -2.1107,E1 25.1548,E2 104.3354} C_DIS
LIN {X 82.6855,Y -22.8807,Z 90,A -20.8092,B 24.9168,C -2.1066,E1 25.1538,E2 105.7069} C_DIS
LIN {X 82.0907,Y -24.93,Z 90,A -22.2122,B 24.9171,C -2.1029,E1 25.1527,E2 107.1107} C_DIS
LIN {X 81.4495,Y -26.9508,Z 90,A -23.6077,B 24.9174,C -2.0992,E1 25.1515,E2 108.5071} C_DIS
LIN {X 80.777,Y -28.9049,Z 90,A -25.0225,B 24.9178,C -2.0937,E1 25.1501,E2 109.9268} C_DIS
LIN {X 79.8435,Y -31.387,Z 90,A -26.8766,B 24.9184,C -2.0855,E1 25.1483,E2 111.7901} C_DIS
LIN {X 78.8444,Y -33.8224,Z 90,A -28.5258,B 24.9186,C -2.0838,E1 25.1465,E2 113.434} C_DIS
LIN {X 77.9789,Y -35.7723,Z 90,A -29.8978,B 24.9188,C -2.0814,E1 25.1449,E2 114.8045} C_DIS
LIN {X 77.0808,Y -37.6684,Z 90,A -31.29,B 24.9191,C -2.0775,E1 25.1433,E2 116.1983} C_DIS
LIN {X 75.973,Y -39.853,Z 90,A -33.0982,B 24.9199,C -2.0668,E1 25.1409,E2 118.0221} C_DIS
LIN {X 74.6529,Y -42.2771,Z 90,A -34.7716,B 24.9199,C -2.0672,E1 25.1387,E2 119.6859} C_DIS
LIN {X 73.597,Y -44.0894,Z 90,A -36.1704,B 24.9202,C -2.0633,E1 25.1367,E2 121.0868} C_DIS
LIN {X 72.484,Y -45.8964,Z 90,A -37.572,B 24.9204,C -2.0598,E1 25.1346,E2 122.4896} C_DIS
LIN {X 71.2961,Y -47.7202,Z 90,A -39.0083,B 24.9207,C -2.0563,E1 25.1324,E2 123.927} C_DIS
LIN {X 70.1351,Y -49.4112,Z 90,A -40.3977,B 24.9211,C -2.0518,E1 25.1302,E2 125.32} C_DIS
LIN {X 68.9055,Y -51.112,Z 90,A -41.9857,B 24.9218,C -2.0417,E1 25.1275,E2 126.9242} C_DIS
LIN {X 66.9835,Y -53.6061,Z 90,A -44.0989,B 24.9223,C -2.0358,E1 25.1239,E2 129.0415} C_DIS
LIN {X 64.9621,Y -56.0387,Z 90,A -46.1886,B 24.9226,C -2.0311,E1 25.1201,E2 131.1328} C_DIS
LIN {X 62.834,Y -58.4146,Z 90,A -48.289,B 24.923,C -2.0267,E1 25.1161,E2 133.2342} C_DIS
LIN {X 60.6513,Y -60.678,Z 90,A -50.3816,B 24.9233,C -2.0219,E1 25.112,E2 135.3294} C_DIS
LIN {X 58.3753,Y -62.8707,Z 90,A -52.4817,B 24.9237,C -2.0172,E1 25.1078,E2 137.4319} C_DIS
LIN {X 56.0128,Y -64.9842,Z 90,A -54.5844,B 24.924,C -2.0129,E1 25.1033,E2 139.5366} C_DIS
LIN {X 53.6055,Y -66.984,Z 90,A -56.671,B 24.9244,C -2.0084,E1 25.0988,E2 141.6258} C_DIS
LIN {X 51.1117,Y -68.9057,Z 90,A -58.5647,B 24.9242,C -2.0109,E1 25.0946,E2 143.5068} C_DIS
LIN {X 49.2616,Y -70.2393,Z 90,A -60.2242,B 24.9248,C -2.0033,E1 25.0908,E2 145.1785} C_DIS
LIN {X 46.7171,Y -71.9572,Z 90,A -62.0804,B 24.9246,C -2.0056,E1 25.0865,E2 147.0229} C_DIS
LIN {X 44.8754,Y -73.1196,Z 90,A -63.5016,B 24.9246,C -2.004,E1 25.0832,E2 148.4435} C_DIS
LIN {X 43.1518,Y -74.1504,Z 90,A -64.8881,B 24.925,C -2,E1 25.0798,E2 149.8351} C_DIS
LIN {X 41.3589,Y -75.1655,Z 90,A -66.2808,B 24.9252,C -1.9971,E1 25.0764,E2 151.2307} C_DIS
LIN {X 39.4586,Y -76.1799,Z 90,A -67.6584,B 24.9252,C -1.9966,E1 25.073,E2 152.6055} C_DIS
LIN {X 37.6029,Y -77.1129,Z 90,A -69.1563,B 24.9257,C -1.9908,E1 25.0693,E2 154.1132} C_DIS
LIN {X 35.7193,Y -78.0034,Z 90,A -70.4847,B 24.9257,C -1.9906,E1 25.0659,E2 155.4385} C_DIS
LIN {X 33.7635,Y -78.8695,Z 90,A -71.8644,B 24.9257,C -1.9901,E1 25.0624,E2 156.8162} C_DIS
LIN {X 31.8542,Y -79.66,Z 90,A -73.2963,B 24.926,C -1.9865,E1 25.0586,E2 158.2535} C_DIS
LIN {X 29.8133,Y -80.4456,Z 90,A -74.7146,B 24.926,C -1.9859,E1 25.0549,E2 159.6701} C_DIS
LIN {X 27.8797,Y -81.1363,Z 90,A -76.1044,B 24.9262,C -1.9835,E1 25.0513,E2 161.0627} C_DIS
LIN {X 25.8917,Y -81.7925,Z 90,A -77.573,B 24.9265,C -1.9795,E1 25.0474,E2 162.5379} C_DIS
LIN {X 23.8514,Y -82.4104,Z 90,A -78.8765,B 24.9264,C -1.9818,E1 25.0439,E2 163.8337} C_DIS
LIN {X 21.8659,Y -82.9596,Z 90,A -80.2934,B 24.9266,C -1.979,E1 25.0401,E2 165.255} C_DIS
LIN {X 19.7973,Y -83.4772,Z 90,A -81.6922,B 24.9266,C -1.9784,E1 25.0363,E2 166.6532} C_DIS
LIN {X 16.6982,Y -84.1519,Z 90,A -83.8087,B 24.9267,C -1.9766,E1 25.0305,E2 168.7713} C_DIS
LIN {X 14.6662,Y -84.53,Z 90,A -85.1874,B 24.9268,C -1.9756,E1 25.0267,E2 170.151} C_DIS
LIN {X 12.2935,Y -84.9062,Z 90,A -86.9493,B 24.9273,C -1.9695,E1 25.0218,E2 171.9257} C_DIS
LIN {X 9.4129,Y -85.2746,Z 90,A -88.7031,B 24.9269,C -1.9741,E1 25.017,E2 173.6671} C_DIS
LIN {X 7.3203,Y -85.4797,Z 90,A -90.321,B 24.9275,C -1.9667,E1 25.0124,E2 175.3018} C_DIS
LIN {X 4.2096,Y -85.6895,Z 90,A -92.2092,B 24.9271,C -1.9719,E1 25.0072,E2 177.1768} C_DIS
LIN {X 2.0718,Y -85.7676,Z 90,A -93.8328,B 24.9276,C -1.9653,E1 25.0026,E2 178.8157} C_DIS
LIN {X 2.0718,Y -85.7676,Z 90,A -93.8328,B 24.9276,C -1.9653,E1 25.0026,E2 178.8157} C_DIS
Enddeposition()
LIN {X 0.6275,Y -93.7513,Z 91,A -93.8852,B 24.9349,C -1.8634,E1 25.0018,E2 179.1097} C_DIS
Startdeposition()
$VEL.CP = VEL_PRINT
LIN {X -1.4988,Y -93.7433,Z 91,A -95.8353,B 24.9365,C -1.8406,E1 24.9962,E2 181.114} C_DIS
LIN {X -5.2351,Y -93.6087,Z 91,A -98.0025,B 24.9362,C -1.8444,E1 24.9902,E2 183.2726} C_DIS
LIN {X -8.4243,Y -93.3759,Z 91,A -100.0173,B 24.9364,C -1.8424,E1 24.9845,E2 185.2931} C_DIS
LIN {X -11.6435,Y -93.03,Z 91,A -102.0393,B 24.9364,C -1.8412,E1 24.9789,E2 187.3193} C_DIS
LIN {X -14.8871,Y -92.5672,Z 91,A -104.077,B 24.9365,C -1.8405,E1 24.9733,E2 189.3604} C_DIS
LIN {X -18.1492,Y -91.9825,Z 91,A -106.0835,B 24.9365,C -1.8419,E1 24.9678,E2 191.3658} C_DIS
LIN {X -21.4236,Y -91.275,Z 91,A -108.0479,B 24.9361,C -1.8457,E1 24.9625,E2 193.3237} C_DIS
LIN {X -24.7039,Y -90.4421,Z 91,A -110.1197,B 24.9361,C -1.8468,E1 24.9569,E2 195.3959} C_DIS
LIN {X -27.8682,Y -89.5174,Z 91,A -112.2065,B 24.9361,C -1.8458,E1 24.9513,E2 197.4887} C_DIS
LIN {X -31.2547,Y -88.3922,Z 91,A -114.3563,B 24.9359,C -1.8486,E1 24.9456,E2 199.6358} C_DIS
LIN {X -34.5108,Y -87.1726,Z 91,A -116.5331,B 24.9359,C -1.8489,E1 24.9399,E2 201.8166} C_DIS
LIN {X -37.7441,Y -85.8223,Z 91,A -118.6917,B 24.9359,C -1.8506,E1 24.9344,E2 203.9762} C_DIS
LIN {X -40.947,Y -84.3414,Z 91,A -120.8687,B 24.9357,C -1.8524,E1 24.9289,E2 206.1544} C_DIS
LIN {X -44.1119,Y -82.7307,Z 91,A -123.0434,B 24.9355,C -1.855,E1 24.9235,E2 208.3288} C_DIS
LIN {X -47.21,Y -81.003,Z 91,A -125.2335,B 24.9353,C -1.8573,E1 24.9182,E2 210.5199} C_DIS
LIN {X -50.0722,Y -79.2653,Z 91,A -127.2744,B 24.9351,C -1.8606,E1 24.9133,E2 212.5595} C_DIS
LIN {X -52.8032,Y -77.4719,Z 91,A -129.2233,B 24.9348,C -1.8653,E1 24.9088,E2 214.5036} C_DIS
LIN {X -55.7508,Y -75.3793,Z 91,A -131.4957,B 24.9347,C -1.867,E1 24.9037,E2 216.78} C_DIS
LIN {X -58.3589,Y -73.3779,Z 91,A -133.5123,B 24.9344,C -1.8704,E1 24.8992,E2 218.7959} C_DIS
LIN {X -61.2391,Y -70.9931,Z 91,A -135.8085,B 24.9341,C -1.8744,E1 24.8943,E2 221.0915} C_DIS
LIN {X -63.6719,Y -68.8188,Z 91,A -137.7085,B 24.9336,C -1.8813,E1 24.8904,E2 222.9825} C_DIS
LIN {X -66.055,Y -66.5341,Z 91,A -139.6843,B 24.9333,C -1.8869,E1 24.8865,E2 224.9533} C_DIS
LIN {X -68.4049,Y -64.1154,Z 91,A -141.8203,B 24.9331,C -1.8889,E1 24.8824,E2 227.0938} C_DIS
LIN {X -70.6651,Y -61.6153,Z 91,A -143.8218,B 24.9327,C -1.8954,E1 24.8787,E2 229.0888} C_DIS
LIN {X -72.787,Y -59.0936,Z 91,A -145.8787,B 24.9324,C -1.8987,E1 24.875,E2 231.1472} C_DIS
LIN {X -74.8578,Y -56.4476,Z 91,A -147.9913,B 24.9322,C -1.9018,E1 24.8714,E2 233.2625} C_DIS
LIN {X -76.9395,Y -53.5753,Z 91,A -150.1206,B 24.9317,C -1.9084,E1 24.8679,E2 235.3866} C_DIS
LIN {X -78.7994,Y -50.8004,Z 91,A -152.2365,B 24.9315,C -1.9113,E1 24.8647,E2 237.5062} C_DIS
LIN {X -80.6872,Y -47.7448,Z 91,A -154.4183,B 24.9311,C -1.9174,E1 24.8615,E2 239.6845} C_DIS
LIN {X -82.4485,Y -44.6345,Z 91,A -156.5876,B 24.9306,C -1.9238,E1 24.8586,E2 241.85} C_DIS
LIN {X -84.0506,Y -41.5391,Z 91,A -158.7648,B 24.9303,C -1.9282,E1 24.8559,E2 244.0284} C_DIS
LIN {X -85.5561,Y -38.3429,Z 91,A -160.987,B 24.93,C -1.9323,E1 24.8533,E2 246.2529} C_DIS
LIN {X -86.931,Y -35.1149,Z 91,A -163.1488,B 24.9296,C -1.938,E1 24.8509,E2 248.4133} C_DIS
LIN {X -88.2213,Y -31.7359,Z 91,A -165.351,B 24.9291,C -1.9447,E1 24.8488,E2 250.612} C_DIS
LIN {X -89.3299,Y -28.4663,Z 91,A -167.4703,B 24.9287,C -1.9507,E1 24.847,E2 252.729} C_DIS
LIN {X -90.3091,Y -25.1875,Z 91,A -169.563,B 24.9282,C -1.9569,E1 24.8453,E2 254.8189} C_DIS
LIN {X -91.1291,Y -22.0343,Z 91,A -171.5241,B 24.9277,C -1.9639,E1 24.844,E2 256.7747} C_DIS
LIN {X -91.8854,Y -18.631,Z 91,A -173.6244,B 24.9271,C -1.9714,E1 24.8428,E2 258.8695} C_DIS
LIN {X -92.4659,Y -15.4933,Z 91,A -175.64,B 24.9268,C -1.9755,E1 24.8418,E2 260.8874} C_DIS
LIN {X -92.9683,Y -12.12,Z 91,A -177.7231,B 24.9263,C -1.9821,E1 24.841,E2 262.9672} C_DIS
LIN {X -93.3208,Y -9.0219,Z 91,A -179.7878,B 24.9263,C -1.9832,E1 24.8404,E2 265.0416} C_DIS
LIN {X -93.6087,Y -5.2351,Z 91,A 177.9533,B 24.9256,C -1.9925,E1 24.84,E2 267.2919} C_DIS
LIN {X -93.7433,Y -1.4988,Z 91,A 175.7942,B 24.9247,C -2.0037,E1 24.8398,E2 269.4374} C_DIS
LIN {X -93.7433,Y 1.4988,Z 91,A 173.7773,B 24.9247,C -2.0039,E1 24.8398,E2 271.4659} C_DIS
LIN {X -93.6087,Y 5.2351,Z 91,A 171.6241,B 24.9239,C -2.0152,E1 24.8401,E2 273.6049} C_DIS
LIN {X -93.3759,Y 8.4243,Z 91,A 169.5654,B 24.9236,C -2.0183,E1 24.8406,E2 275.6687} C_DIS
LIN {X -93.03,Y 11.6435,Z 91,A 167.5297,B 24.9233,C -2.0229,E1 24.8412,E2 277.7057} C_DIS
LIN {X -92.5672,Y 14.8871,Z 91,A 165.4785,B 24.9229,C -2.0278,E1 24.8421,E2 279.7574} C_DIS
LIN {X -91.9825,Y 18.1492,Z 91,A 163.4597,B 24.9224,C -2.0344,E1 24.8431,E2 281.7723} C_DIS
LIN {X -91.275,Y 21.4236,Z 91,A 161.4837,B 24.9217,C -2.0431,E1 24.8443,E2 283.7392} C_DIS
LIN {X -90.4421,Y 24.7039,Z 91,A 159.3733,B 24.9213,C -2.0483,E1 24.8458,E2 285.8494} C_DIS
LIN {X -89.4817,Y 27.9834,Z 91,A 157.2298,B 24.9209,C -2.0532,E1 24.8476,E2 287.9936} C_DIS
LIN {X -88.3922,Y 31.2547,Z 91,A 155.1416,B 24.9204,C -2.0603,E1 24.8494,E2 290.0768} C_DIS
LIN {X -87.1726,Y 34.5108,Z 91,A 152.9543,B 24.92,C -2.0649,E1 24.8516,E2 292.2654} C_DIS
LIN {X -85.8223,Y 37.7441,Z 91,A 150.7864,B 24.9196,C -2.0705,E1 24.854,E2 294.4318} C_DIS
LIN {X -84.3414,Y 40.947,Z 91,A 148.6005,B 24.9192,C -2.0761,E1 24.8566,E2 296.6164} C_DIS
LIN {X -82.7371,Y 44.0997,Z 91,A 146.4249,B 24.9187,C -2.082,E1 24.8594,E2 298.7895} C_DIS
LIN {X -81.003,Y 47.21,Z 91,A 144.2207,B 24.9183,C -2.0874,E1 24.8625,E2 300.9924} C_DIS
LIN {X -79.2653,Y 50.0722,Z 91,A 142.1737,B 24.9178,C -2.0931,E1 24.8655,E2 303.036} C_DIS
LIN {X -77.4719,Y 52.8032,Z 91,A 140.1919,B 24.9174,C -2.0991,E1 24.8686,E2 305.0134} C_DIS
LIN {X -75.3793,Y 55.7508,Z 91,A 137.9422,B 24.917,C -2.1039,E1 24.8723,E2 307.2628} C_DIS
LIN {X -73.3779,Y 58.3589,Z 91,A 135.9218,B 24.9166,C -2.1088,E1 24.8757,E2 309.2808} C_DIS
LIN {X -70.9931,Y 61.2391,Z 91,A 133.6223,B 24.9162,C -2.1143,E1 24.8799,E2 311.578} C_DIS
LIN {X -68.8188,Y 63.6719,Z 91,A 131.7202,B 24.9155,C -2.1221,E1 24.8834,E2 313.4698} C_DIS
LIN {X -66.5341,Y 66.055,Z 91,A 129.7427,B 24.915,C -2.1283,E1 24.8873,E2 315.441} C_DIS
LIN {X -64.1154,Y 68.4049,Z 91,A 127.6059,B 24.9148,C -2.1308,E1 24.8916,E2 317.5808} C_DIS
LIN {X -61.6153,Y 70.6651,Z 91,A 125.6042,B 24.9143,C -2.1373,E1 24.8958,E2 319.575} C_DIS
LIN {X -59.0936,Y 72.787,Z 91,A 123.5479,B 24.9141,C -2.1404,E1 24.9002,E2 321.6317} C_DIS
LIN {X -56.7171,Y 74.6553,Z 91,A 121.5651,B 24.9141,C -2.14,E1 24.9046,E2 323.6227} C_DIS
LIN {X -53.7936,Y 76.7878,Z 91,A 119.4344,B 24.9135,C -2.147,E1 24.9094,E2 325.744} C_DIS
LIN {X -51.304,Y 78.4731,Z 91,A 117.5185,B 24.9135,C -2.1481,E1 24.9139,E2 327.6638} C_DIS
LIN {X -48.2588,Y 80.3825,Z 91,A 115.2925,B 24.9132,C -2.1512,E1 24.9192,E2 329.8892} C_DIS
LIN {X -45.157,Y 82.1651,Z 91,A 113.0853,B 24.913,C -2.1543,E1 24.9245,E2 332.0954} C_DIS
LIN {X -42.1534,Y 83.7444,Z 91,A 111.0312,B 24.9126,C -2.1584,E1 24.9296,E2 334.1455} C_DIS
LIN {X -38.8155,Y 85.3432,Z 91,A 108.7796,B 24.9123,C -2.1621,E1 24.9353,E2 336.3937} C_DIS
LIN {X -35.5915,Y 86.737,Z 91,A 106.6412,B 24.912,C -2.1655,E1 24.9408,E2 338.5291} C_DIS
LIN {X -32.3422,Y 88.0002,Z 91,A 104.5141,B 24.9118,C -2.1684,E1 24.9464,E2 340.6537} C_DIS
LIN {X -29.0751,Y 89.133,Z 91,A 102.3991,B 24.9116,C -2.1709,E1 24.9519,E2 342.7668} C_DIS
LIN {X -25.7975,Y 90.1362,Z 91,A 100.2971,B 24.9114,C -2.1729,E1 24.9576,E2 344.8674} C_DIS
LIN {X -22.6744,Y 90.972,Z 91,A 98.2698,B 24.9114,C -2.1732,E1 24.9631,E2 346.897} C_DIS
LIN {X -18.929,Y 91.8242,Z 91,A 95.9894,B 24.9111,C -2.1775,E1 24.9693,E2 349.1701} C_DIS
LIN {X -15.4933,Y 92.4659,Z 91,A 93.8752,B 24.9109,C -2.1798,E1 24.9751,E2 351.2809} C_DIS
LIN {X -12.12,Y 92.9683,Z 91,A 91.8036,B 24.9107,C -2.1815,E1 24.9808,E2 353.35} C_DIS
LIN {X -9.0219,Y 93.3208,Z 91,A 89.7508,B 24.9111,C -2.1776,E1 24.9865,E2 355.4133} C_DIS
LIN {X -5.2351,Y 93.6087,Z 91,A 87.5056,B 24.9108,C -2.1811,E1 24.9927,E2 357.651} C_DIS
LIN {X -1.4988,Y 93.7433,Z 91,A 85.3493,B 24.9104,C -2.1861,E1 24.9987,E2 359.7958} C_DIS
LIN {X 1.4988,Y 93.7433,Z 91,A 83.3569,B 24.9108,C -2.181,E1 25.0043,E2 361.8} C_DIS
LIN {X 5.2351,Y 93.6087,Z 91,A 81.1892,B 24.9104,C -2.1851,E1 25.0103,E2 363.9574} C_DIS
LIN {X 8.4243,Y 93.3759,Z 91,A 79.1748,B 24.9106,C -2.1829,E1 25.016,E2 365.976} C_DIS
LIN {X 11.6435,Y 93.03,Z 91,A 77.1541,B 24.9108,C -2.1811,E1 25.0216,E2 367.9994} C_DIS
LIN {X 14.8326,Y 92.5756,Z 91,A 75.1481,B 24.9109,C -2.1793,E1 25.0271,E2 370.0079} C_DIS
LIN {X 18.1492,Y 91.9825,Z 91,A 73.1144,B 24.9109,C -2.1793,E1 25.0327,E2 372.0392} C_DIS
LIN {X 21.4236,Y 91.275,Z 91,A 71.1557,B 24.9108,C -2.1813,E1 25.038,E2 373.9905} C_DIS
LIN {X 24.7039,Y 90.4421,Z 91,A 69.0628,B 24.9109,C -2.1792,E1 25.0437,E2 376.0852} C_DIS
LIN {X 27.9834,Y 89.4817,Z 91,A 66.9373,B 24.9112,C -2.1763,E1 25.0494,E2 378.2136} C_DIS
LIN {X 31.2547,Y 88.3922,Z 91,A 64.8291,B 24.9113,C -2.1745,E1 25.0549,E2 380.322} C_DIS
LIN {X 34.5108,Y 87.1726,Z 91,A 62.6995,B 24.9115,C -2.1723,E1 25.0605,E2 382.4523} C_DIS
LIN {X 37.7441,Y 85.8223,Z 91,A 60.551,B 24.9117,C -2.1697,E1 25.066,E2 384.6017} C_DIS
LIN {X 40.947,Y 84.3414,Z 91,A 58.3852,B 24.9119,C -2.1668,E1 25.0715,E2 386.7687} C_DIS
LIN {X 44.0997,Y 82.7371,Z 91,A 56.2297,B 24.9122,C -2.1642,E1 25.0768,E2 388.9245} C_DIS
LIN {X 47.21,Y 81.003,Z 91,A 54.0463,B 24.9124,C -2.1609,E1 25.0821,E2 391.1092} C_DIS
LIN {X 50.0722,Y 79.2653,Z 91,A 52.0188,B 24.9126,C -2.1584,E1 25.0869,E2 393.1361} C_DIS
LIN {X 52.8032,Y 77.4719,Z 91,A 50.0558,B 24.9128,C -2.1564,E1 25.0915,E2 395.0973} C_DIS
LIN {X 55.7508,Y 75.3793,Z 91,A 47.8282,B 24.9131,C -2.1519,E1 25.0965,E2 397.3276} C_DIS
LIN {X 58.3589,Y 73.3779,Z 91,A 45.8275,B 24.9134,C -2.1486,E1 25.1009,E2 399.3288} C_DIS
LIN {X 61.2391,Y 70.9931,Z 91,A 43.5505,B 24.9137,C -2.1445,E1 25.1058,E2 401.6067} C_DIS
LIN {X 63.6719,Y 68.8188,Z 91,A 41.6672,B 24.9137,C -2.1445,E1 25.1096,E2 403.4825} C_DIS
LIN {X 66.055,Y 66.5341,Z 91,A 39.7092,B 24.9139,C -2.1424,E1 25.1135,E2 405.4371} C_DIS
LIN {X 68.4049,Y 64.1154,Z 91,A 37.5935,B 24.9144,C -2.1359,E1 25.1176,E2 407.5589} C_DIS
LIN {X 70.6651,Y 61.6153,Z 91,A 35.6118,B 24.9146,C -2.1341,E1 25.1213,E2 409.5362} C_DIS
LIN {X 72.787,Y 59.0936,Z 91,A 33.5759,B 24.915,C -2.1286,E1 25.1249,E2 411.5756} C_DIS
LIN {X 74.8578,Y 56.4476,Z 91,A 31.4857,B 24.9155,C -2.1223,E1 25.1285,E2 413.6709} C_DIS
LIN {X 76.9395,Y 53.5753,Z 91,A 29.3791,B 24.9158,C -2.1191,E1 25.1319,E2 415.7746} C_DIS
LIN {X 78.7994,Y 50.8004,Z 91,A 27.2872,B 24.9163,C -2.112,E1 25.1351,E2 417.8729} C_DIS
LIN {X 80.6872,Y 47.7448,Z 91,A 25.1302,B 24.9167,C -2.1077,E1 25.1383,E2 420.0292} C_DIS
LIN {X 82.4485,Y 44.6345,Z 91,A 22.9639,B 24.9171,C -2.1024,E1 25.1412,E2 422.1966} C_DIS
LIN {X 84.0506,Y 41.5391,Z 91,A 20.8358,B 24.9176,C -2.0966,E1 25.1439,E2 424.3272} C_DIS
LIN {X 85.5561,Y 38.3429,Z 91,A 18.6853,B 24.918,C -2.0908,E1 25.1464,E2 426.4797} C_DIS
LIN {X 86.931,Y 35.1149,Z 91,A 16.6021,B 24.9183,C -2.0869,E1 25.1486,E2 428.5607} C_DIS
LIN {X 88.1311,Y 31.9833,Z 91,A 14.4427,B 24.9191,C -2.0768,E1 25.1508,E2 430.7319} C_DIS
LIN {X 89.3299,Y 28.4663,Z 91,A 12.2403,B 24.9194,C -2.0726,E1 25.1527,E2 432.9317} C_DIS
LIN {X 90.3091,Y 25.1875,Z 91,A 10.1752,B 24.9199,C -2.0672,E1 25.1543,E2 434.9977} C_DIS
LIN {X 91.1291,Y 22.0343,Z 91,A 8.2403,B 24.9202,C -2.0632,E1 25.1556,E2 436.9308} C_DIS
LIN {X 91.8467,Y 18.8197,Z 91,A 6.2394,B 24.9206,C -2.0574,E1 25.1568,E2 438.9337} C_DIS
LIN {X 92.466,Y 15.4933,Z 91,A 4.1886,B 24.9211,C -2.0516,E1 25.1578,E2 440.9862} C_DIS
LIN {X 92.9683,Y 12.12,Z 91,A 2.0479,B 24.9217,C -2.043,E1 25.1586,E2 443.1348} C_DIS
LIN {X 93.3759,Y 8.4243,Z 91,A -0.0918,B 24.9219,C -2.0407,E1 25.1592,E2 445.2671} C_DIS
LIN {X 93.6087,Y 5.2351,Z 91,A -2.1381,B 24.9226,C -2.031,E1 25.1596,E2 447.3241} C_DIS
LIN {X 93.7433,Y 1.4988,Z 91,A -4.2672,B 24.9228,C -2.0295,E1 25.1598,E2 449.4441} C_DIS
LIN {X 93.7433,Y -1.4988,Z 91,A -6.2557,B 24.9237,C -2.0178,E1 25.1598,E2 451.4484} C_DIS
LIN {X 93.6087,Y -5.2351,Z 91,A -8.4081,B 24.9238,C -2.0154,E1 25.1595,E2 453.5937} C_DIS
LIN {X 93.3759,Y -8.4243,Z 91,A -10.4087,B 24.9244,C -2.0074,E1 25.159,E2 455.6013} C_DIS
LIN {X 93.03,Y -11.6435,Z 91,A -12.4159,B 24.925,C -1.9999,E1 25.1584,E2 457.6142} C_DIS
LIN {X 92.5672,Y -14.8871,Z 91,A -14.4382,B 24.9255,C -1.9928,E1 25.1575,E2 459.6415} C_DIS
LIN {X 91.9825,Y -18.1492,Z 91,A -16.4291,B 24.9259,C -1.9876,E1 25.1565,E2 461.6331} C_DIS
LIN {X 91.275,Y -21.4236,Z 91,A -18.3779,B 24.9261,C -1.9848,E1 25.1553,E2 463.5771} C_DIS
LIN {X 90.4421,Y -24.7039,Z 91,A -20.4592,B 24.9267,C -1.9778,E1 25.1538,E2 465.663} C_DIS
LIN {X 89.4817,Y -27.9834,Z 91,A -22.5657,B 24.9272,C -1.9705,E1 25.1521,E2 467.7745} C_DIS
LIN {X 88.3922,Y -31.2547,Z 91,A -24.6335,B 24.9276,C -1.9655,E1 25.1502,E2 469.8427} C_DIS
LIN {X 87.1726,Y -34.5108,Z 91,A -26.7912,B 24.9281,C -1.9577,E1 25.1481,E2 472.0067} C_DIS
LIN {X 85.8223,Y -37.7441,Z 91,A -28.9305,B 24.9286,C -1.9513,E1 25.1457,E2 474.1495} C_DIS
LIN {X 84.3414,Y -40.947,Z 91,A -31.0878,B 24.9291,C -1.9448,E1 25.1431,E2 476.3105} C_DIS
LIN {X 82.7435,Y -44.0876,Z 91,A -33.229,B 24.9295,C -1.9389,E1 25.1403,E2 478.4543} C_DIS
LIN {X 81.003,Y -47.21,Z 91,A -35.412,B 24.93,C -1.9326,E1 25.1373,E2 480.6408} C_DIS
LIN {X 79.2653,Y -50.0722,Z 91,A -37.4336,B 24.9303,C -1.9277,E1 25.1343,E2 482.6637} C_DIS
LIN {X 77.4719,Y -52.8032,Z 91,A -39.2655,B 24.9303,C -1.9282,E1 25.1315,E2 484.4853} C_DIS
LIN {X 75.5783,Y -55.479,Z 91,A -41.2869,B 24.9307,C -1.9221,E1 25.1282,E2 486.5113} C_DIS
LIN {X 73.5435,Y -58.1494,Z 91,A -43.3857,B 24.9313,C -1.9149,E1 25.1246,E2 488.6173} C_DIS
LIN {X 71.2363,Y -60.9542,Z 91,A -45.6211,B 24.9317,C -1.9085,E1 25.1206,E2 490.8576} C_DIS
LIN {X 68.9082,Y -63.5745,Z 91,A -47.7087,B 24.932,C -1.9051,E1 25.1167,E2 492.9439} C_DIS
LIN {X 66.5341,Y -66.055,Z 91,A -49.7225,B 24.9321,C -1.903,E1 25.1128,E2 494.954} C_DIS
LIN {X 64.1154,Y -68.4049,Z 91,A -51.8374,B 24.9326,C -1.8961,E1 25.1085,E2 497.0763} C_DIS
LIN {X 61.6153,Y -70.6651,Z 91,A -53.819,B 24.9327,C -1.8942,E1 25.1044,E2 499.0545} C_DIS
LIN {X 59.0936,Y -72.787,Z 91,A -55.8555,B 24.9331,C -1.8889,E1 25.1,E2 501.0957} C_DIS
LIN {X 56.4476,Y -74.8578,Z 91,A -57.947,B 24.9335,C -1.8831,E1 25.0953,E2 503.1933} C_DIS
LIN {X 53.5753,Y -76.9395,Z 91,A -60.0553,B 24.9337,C -1.8809,E1 25.0905,E2 505.2996} C_DIS
LIN {X 50.8004,Y -78.7994,Z 91,A -62.1503,B 24.9341,C -1.8749,E1 25.0856,E2 507.4016} C_DIS
LIN {X 47.7448,Y -80.6872,Z 91,A -64.3108,B 24.9343,C -1.8721,E1 25.0805,E2 509.5621} C_DIS
LIN {X 44.6345,Y -82.4485,Z 91,A -66.4589,B 24.9345,C -1.8696,E1 25.0752,E2 511.7099} C_DIS
LIN {X 41.5391,Y -84.0506,Z 91,A -68.6151,B 24.9348,C -1.8651,E1 25.0699,E2 513.8707} C_DIS
LIN {X 38.3724,Y -85.5428,Z 91,A -70.8039,B 24.9351,C -1.86,E1 25.0643,E2 516.0661} C_DIS
LIN {X 35.1149,Y -86.931,Z 91,A -72.9573,B 24.9353,C -1.8573,E1 25.0587,E2 518.2211} C_DIS
LIN {X 31.7359,Y -88.2213,Z 91,A -75.1391,B 24.9355,C -1.8553,E1 25.053,E2 520.4028} C_DIS
LIN {X 28.4663,Y -89.3299,Z 91,A -77.2388,B 24.9356,C -1.8531,E1 25.0475,E2 522.5038} C_DIS
LIN {X 25.1875,Y -90.3091,Z 91,A -79.3126,B 24.9357,C -1.8514,E1 25.0419,E2 524.5781} C_DIS
LIN {X 22.0343,Y -91.1291,Z 91,A -81.2563,B 24.9357,C -1.8511,E1 25.0366,E2 526.5196} C_DIS
LIN {X 18.631,Y -91.8854,Z 91,A -83.3384,B 24.9357,C -1.8509,E1 25.031,E2 528.5995} C_DIS
LIN {X 15.4933,Y -92.4659,Z 91,A -85.3367,B 24.936,C -1.8476,E1 25.0254,E2 530.6033} C_DIS
LIN {X 12.12,Y -92.9683,Z 91,A -87.4023,B 24.936,C -1.8469,E1 25.0197,E2 532.6689} C_DIS
LIN {X 9.0219,Y -93.3208,Z 91,A -89.45,B 24.9365,C -1.8408,E1 25.014,E2 534.7296} C_DIS
LIN {X 5.2351,Y -93.6087,Z 91,A -91.6911,B 24.9364,C -1.8426,E1 25.0078,E2 536.9655} C_DIS
LIN {X 1.4988,Y -93.7433,Z 91,A -93.8446,B 24.9361,C -1.8464,E1 25.0018,E2 539.1096} C_DIS
LIN {X 1.4988,Y -93.7433,Z 91,A -93.8446,B 24.9361,C -1.8464,E1 25.0018,E2 539.1096} C_DIS
Enddeposition()
LIN {X 0.633,Y -92.7825,Z 91,A -94.7091,B 24.9357,C -1.8519,E1 24.9994,E2 539.961} C_DIS
Startdeposition()
$VEL.CP = VEL_PRINT
LIN {X 4.9066,Y -92.6575,Z 91,A -90.5583,B 24.932,C -1.9049,E1 25.0114,E2 535.6854} C_DIS
LIN {X 9.6744,Y -92.2813,Z 91,A -87.7409,B 24.9322,C -1.9017,E1 25.0192,E2 532.8774} C_DIS
LIN {X 14.8397,Y -91.5938,Z 91,A -84.4762,B 24.9319,C -1.9056,E1 25.0282,E2 529.6064} C_DIS
LIN {X 19.1844,Y -90.7824,Z 91,A -82.0383,B 24.9325,C -1.8976,E1 25.0348,E2 527.1904} C_DIS
LIN {X 22.7125,Y -89.9648,Z 91,A -79.982,B 24.9328,C -1.8934,E1 25.0404,E2 525.147} C_DIS
LIN {X 24.7014,Y -89.4388,Z 91,A -78.2479,B 24.9315,C -1.9112,E1 25.0451,E2 523.3734} C_DIS
LIN {X 29.0236,Y -88.1308,Z 91,A -75.7299,B 24.932,C -1.9049,E1 25.0518,E2 520.8751} C_DIS
LIN {X 32.5353,Y -86.896,Z 91,A -73.7885,B 24.9327,C -1.8951,E1 25.0568,E2 518.9609} C_DIS
LIN {X 37.3105,Y -84.9553,Z 91,A -70.3555,B 24.9317,C -1.9086,E1 25.0658,E2 515.5039} C_DIS
LIN {X 40.9242,Y -83.2743,Z 91,A -67.8261,B 24.9313,C -1.915,E1 25.0721,E2 512.966} C_DIS
LIN {X 43.44,Y -81.9906,Z 91,A -66.0614,B 24.931,C -1.9186,E1 25.0765,E2 511.1975} C_DIS
LIN {X 45.661,Y -80.7759,Z 91,A -63.9863,B 24.9294,C -1.9401,E1 25.0817,E2 509.0778} C_DIS
LIN {X 48.7974,Y -78.9204,Z 91,A -61.7524,B 24.9292,C -1.9437,E1 25.087,E2 506.8424} C_DIS
LIN {X 51.8216,Y -76.9676,Z 91,A -60.2033,B 24.9306,C -1.9234,E1 25.0904,E2 505.3465} C_DIS
LIN {X 55.48,Y -74.3741,Z 91,A -57.2583,B 24.9298,C -1.9355,E1 25.0971,E2 502.3832} C_DIS
LIN {X 58.5268,Y -72.0005,Z 91,A -54.9127,B 24.9295,C -1.9393,E1 25.1023,E2 500.0374} C_DIS
LIN {X 61.33,Y -69.6292,Z 91,A -52.7921,B 24.9295,C -1.939,E1 25.1067,E2 497.9259} C_DIS
LIN {X 63.9924,Y -67.1902,Z 91,A -50.3247,B 24.9285,C -1.9531,E1 25.1118,E2 495.4353} C_DIS
LIN {X 66.9072,Y -64.2875,Z 91,A -47.9233,B 24.9285,C -1.9541,E1 25.1165,E2 493.0417} C_DIS
LIN {X 69.3508,Y -61.6442,Z 91,A -45.9478,B 24.9287,C -1.9506,E1 25.1202,E2 491.0833} C_DIS
LIN {X 71.7706,Y -58.8092,Z 91,A -43.2943,B 24.9273,C -1.9697,E1 25.125,E2 488.3969} C_DIS
LIN {X 75.9209,Y -53.344,Z 91,A -39.4972,B 24.9276,C -1.9647,E1 25.1313,E2 484.6297} C_DIS
LIN {X 78.9369,Y -48.771,Z 91,A -35.837,B 24.9262,C -1.9845,E1 25.1369,E2 480.9411} C_DIS
LIN {X 80.6175,Y -45.9387,Z 91,A -33.8153,B 24.9258,C -1.9899,E1 25.1397,E2 478.917} C_DIS
LIN {X 82.2256,Y -42.9932,Z 91,A -31.0698,B 24.9234,C -2.0214,E1 25.1434,E2 476.1117} C_DIS
LIN {X 84.1183,Y -39.1605,Z 91,A -29.4736,B 24.9257,C -1.99,E1 25.1452,E2 474.5982} C_DIS
LIN {X 85.2844,Y -36.552,Z 91,A -27.3531,B 24.9243,C -2.0087,E1 25.1476,E2 472.4452} C_DIS
LIN {X 86.6848,Y -33.0943,Z 91,A -25.1346,B 24.9241,C -2.0125,E1 25.1499,E2 470.2299} C_DIS
LIN {X 88.1225,Y -29.0486,Z 91,A -22.4975,B 24.9235,C -2.0202,E1 25.1523,E2 467.5894} C_DIS
LIN {X 89.207,Y -25.5265,Z 91,A -20.2574,B 24.923,C -2.026,E1 25.154,E2 465.3485} C_DIS
LIN {X 89.9906,Y -22.6093,Z 91,A -17.9791,B 24.9214,C -2.0475,E1 25.1556,E2 463.0325} C_DIS
LIN {X 91.3169,Y -16.4517,Z 91,A -14.5444,B 24.9218,C -2.0427,E1 25.1575,E2 459.6292} C_DIS
LIN {X 92.1086,Y -11.2025,Z 91,A -11.2248,B 24.9208,C -2.0548,E1 25.1588,E2 456.3007} C_DIS
LIN {X 92.4911,Y -7.4047,Z 91,A -8.9539,B 24.9205,C -2.0591,E1 25.1594,E2 454.0331} C_DIS
LIN {X 92.7162,Y -3.6407,Z 91,A -6.9041,B 24.9207,C -2.0561,E1 25.1597,E2 452.0026} C_DIS
LIN {X 92.7875,Y 0.0739,Z 91,A -4.6,B 24.9201,C -2.0638,E1 25.1597,E2 449.6939} C_DIS
LIN {X 92.6464,Y 5.1072,Z 91,A -1.26,B 24.9187,C -2.0824,E1 25.1595,E2 446.3299} C_DIS
LIN {X 92.2784,Y 9.6936,Z 91,A 1.6254,B 24.9178,C -2.0931,E1 25.1587,E2 443.4364} C_DIS
LIN {X 91.7734,Y 13.676,Z 91,A 4.3403,B 24.9165,C -2.1098,E1 25.1577,E2 440.6982} C_DIS
LIN {X 91.1565,Y 17.3194,Z 91,A 6.4578,B 24.9165,C -2.1107,E1 25.1566,E2 438.5909} C_DIS
LIN {X 90.3142,Y 21.2802,Z 91,A 8.8351,B 24.9162,C -2.1138,E1 25.1552,E2 436.2201} C_DIS
LIN {X 89.4721,Y 24.581,Z 91,A 10.9081,B 24.9158,C -2.119,E1 25.1537,E2 434.1467} C_DIS
LIN {X 88.3535,Y 28.3399,Z 91,A 13.3123,B 24.9153,C -2.1257,E1 25.1517,E2 431.7406} C_DIS
LIN {X 87.1831,Y 31.7576,Z 91,A 15.5617,B 24.9147,C -2.1329,E1 25.1496,E2 429.4866} C_DIS
LIN {X 85.8337,Y 35.2422,Z 91,A 18.6839,B 24.9117,C -2.1702,E1 25.1462,E2 426.2937} C_DIS
LIN {X 83.8693,Y 39.6909,Z 91,A 20.8217,B 24.9136,C -2.1462,E1 25.1438,E2 424.224} C_DIS
LIN {X 82.0941,Y 43.2435,Z 91,A 23.2147,B 24.9132,C -2.1508,E1 25.1407,E2 421.8329} C_DIS
LIN {X 80.4253,Y 46.2732,Z 91,A 25.3455,B 24.9128,C -2.1564,E1 25.1378,E2 419.7} C_DIS
LIN {X 78.5571,Y 49.379,Z 91,A 27.6167,B 24.9122,C -2.1634,E1 25.1345,E2 417.4236} C_DIS
LIN {X 76.587,Y 52.3834,Z 91,A 29.9737,B 24.9113,C -2.1742,E1 25.1308,E2 415.0529} C_DIS
LIN {X 74.1771,Y 55.7422,Z 91,A 32.2567,B 24.9116,C -2.1706,E1 25.127,E2 412.7895} C_DIS
LIN {X 72.0583,Y 58.4555,Z 91,A 34.4243,B 24.9111,C -2.1772,E1 25.1233,E2 410.6164} C_DIS
LIN {X 70.3282,Y 60.5277,Z 91,A 36.5531,B 24.9094,C -2.1979,E1 25.1193,E2 408.4483} C_DIS
LIN {X 68.1114,Y 63.0105,Z 91,A 38.1442,B 24.9104,C -2.1855,E1 25.1164,E2 406.8935} C_DIS
LIN {X 65.5932,Y 65.6297,Z 91,A 40.1809,B 24.9106,C -2.1828,E1 25.1124,E2 404.8719} C_DIS
LIN {X 62.5314,Y 68.5517,Z 91,A 42.9952,B 24.9096,C -2.1954,E1 25.1067,E2 402.0393} C_DIS
LIN {X 59.8686,Y 70.8897,Z 91,A 45.1466,B 24.9094,C -2.1983,E1 25.1021,E2 399.8895} C_DIS
LIN {X 57.2827,Y 72.9948,Z 91,A 47.2048,B 24.909,C -2.2021,E1 25.0976,E2 397.8301} C_DIS
LIN {X 54.7238,Y 74.9317,Z 91,A 49.2389,B 24.9086,C -2.2074,E1 25.093,E2 395.7906} C_DIS
LIN {X 51.4989,Y 77.1853,Z 91,A 51.6726,B 24.9083,C -2.2115,E1 25.0874,E2 393.3554} C_DIS
LIN {X 48.2952,Y 79.2277,Z 91,A 53.9207,B 24.9083,C -2.2117,E1 25.0821,E2 391.1142} C_DIS
LIN {X 45.3081,Y 80.973,Z 91,A 55.6713,B 24.9091,C -2.2011,E1 25.078,E2 389.394} C_DIS
LIN {X 40.4966,Y 83.4833,Z 91,A 59.4243,B 24.9076,C -2.2195,E1 25.0686,E2 385.6077} C_DIS
LIN {X 37.1309,Y 85.0338,Z 91,A 61.6878,B 24.9075,C -2.2212,E1 25.0628,E2 383.3457} C_DIS
LIN {X 33.9208,Y 86.3645,Z 91,A 63.8228,B 24.9073,C -2.223,E1 25.0573,E2 381.2113} C_DIS
LIN {X 30.7687,Y 87.537,Z 91,A 65.8762,B 24.9073,C -2.2241,E1 25.0519,E2 379.1596} C_DIS
LIN {X 27.4277,Y 88.6407,Z 91,A 68.175,B 24.9067,C -2.2302,E1 25.0457,E2 376.8506} C_DIS
LIN {X 23.7098,Y 89.7071,Z 91,A 70.216,B 24.9076,C -2.2197,E1 25.0403,E2 374.8378} C_DIS
LIN {X 20.6917,Y 90.4507,Z 91,A 72.6148,B 24.9061,C -2.2373,E1 25.0337,E2 372.4006} C_DIS
LIN {X 16.576,Y 91.2946,Z 91,A 74.9415,B 24.9068,C -2.2292,E1 25.0274,E2 370.0959} C_DIS
LIN {X 13.761,Y 91.7619,Z 91,A 77.2875,B 24.9051,C -2.2497,E1 25.0208,E2 367.7033} C_DIS
LIN {X 10.1099,Y 92.235,Z 91,A 79.5764,B 24.905,C -2.2506,E1 25.0144,E2 365.4139} C_DIS
LIN {X 6.3759,Y 92.5677,Z 91,A 81.3626,B 24.9065,C -2.2326,E1 25.0096,E2 363.6712} C_DIS
LIN {X 3.9208,Y 92.7042,Z 91,A 83.8394,B 24.9037,C -2.2653,E1 25.0025,E2 361.1176} C_DIS
LIN {X -1.3591,Y 92.7774,Z 91,A 86.1339,B 24.9066,C -2.2316,E1 24.9962,E2 358.903} C_DIS
LIN {X -6.6096,Y 92.552,Z 91,A 89.4003,B 24.9066,C -2.2311,E1 24.9871,E2 355.6369} C_DIS
LIN {X -13.6436,Y 91.7799,Z 91,A 93.7874,B 24.9068,C -2.2291,E1 24.975,E2 351.2515} C_DIS
LIN {X -17.3099,Y 91.1583,Z 91,A 96.1514,B 24.9068,C -2.2296,E1 24.9685,E2 348.8839} C_DIS
LIN {X -20.9609,Y 90.3885,Z 91,A 98.3336,B 24.9073,C -2.2236,E1 24.9626,E2 346.7133} C_DIS
LIN {X -24.3546,Y 89.5339,Z 91,A 100.5343,B 24.9073,C -2.2227,E1 24.9566,E2 344.5114} C_DIS
LIN {X -28.1541,Y 88.4128,Z 91,A 103.251,B 24.9068,C -2.2288,E1 24.9493,E2 341.7754} C_DIS
LIN {X -33.7259,Y 86.441,Z 91,A 106.6425,B 24.9079,C -2.2157,E1 24.9405,E2 338.4083} C_DIS
LIN {X -36.563,Y 85.2796,Z 91,A 108.5737,B 24.908,C -2.2142,E1 24.9355,E2 336.4761} C_DIS
LIN {X -40.0499,Y 83.6986,Z 91,A 110.8351,B 24.9086,C -2.2073,E1 24.9298,E2 334.2256} C_DIS
LIN {X -43.1727,Y 82.1314,Z 91,A 113.0448,B 24.9088,C -2.2054,E1 24.9243,E2 332.0143} C_DIS
LIN {X -48.2514,Y 79.2543,Z 91,A 116.6748,B 24.9092,C -2.1998,E1 24.9156,E2 328.3869} C_DIS
LIN {X -50.2482,Y 78.0037,Z 91,A 118.4027,B 24.9087,C -2.2058,E1 24.9115,E2 326.6391} C_DIS
LIN {X -54.1121,Y 75.375,Z 91,A 121.1355,B 24.9096,C -2.1951,E1 24.9052,E2 323.9224} C_DIS
LIN {X -57.3325,Y 72.9554,Z 91,A 123.5019,B 24.9104,C -2.186,E1 24.9,E2 321.569} C_DIS
LIN {X -60.0513,Y 70.7341,Z 91,A 125.5984,B 24.9109,C -2.179,E1 24.8956,E2 319.4813} C_DIS
LIN {X -62.6208,Y 68.4696,Z 91,A 127.9036,B 24.9109,C -2.1802,E1 24.8907,E2 317.1641} C_DIS
LIN {X -65.4044,Y 65.8163,Z 91,A 130.1997,B 24.9115,C -2.1721,E1 24.8862,E2 314.8777} C_DIS
LIN {X -67.8506,Y 63.292,Z 91,A 132.3405,B 24.912,C -2.1658,E1 24.8821,E2 312.7426} C_DIS
LIN {X -70.3133,Y 60.5452,Z 91,A 134.8702,B 24.9118,C -2.1679,E1 24.8774,E2 310.1965} C_DIS
LIN {X -72.8808,Y 57.4269,Z 91,A 137.1852,B 24.9128,C -2.1558,E1 24.8733,E2 307.8996} C_DIS
LIN {X -74.8534,Y 54.8307,Z 91,A 139.3017,B 24.913,C -2.1536,E1 24.8698,E2 305.7782} C_DIS
LIN {X -76.9264,Y 51.8824,Z 91,A 142.3486,B 24.9114,C -2.1732,E1 24.865,E2 302.6693} C_DIS
LIN {X -79.5485,Y 47.7672,Z 91,A 144.5127,B 24.9143,C -2.138,E1 24.8619,E2 300.578} C_DIS
LIN {X -81.3191,Y 44.6866,Z 91,A 146.7493,B 24.9147,C -2.133,E1 24.8589,E2 298.3417} C_DIS
LIN {X -83.0104,Y 41.4583,Z 91,A 149.0011,B 24.9152,C -2.1264,E1 24.856,E2 296.0935} C_DIS
LIN {X -84.5397,Y 38.2426,Z 91,A 150.8798,B 24.9165,C -2.11,E1 24.8538,E2 294.2437} C_DIS
LIN {X -85.9194,Y 35.0329,Z 91,A 153.3252,B 24.9163,C -2.1123,E1 24.8511,E2 291.7792} C_DIS
LIN {X -86.7312,Y 32.972,Z 91,A 155.0159,B 24.9159,C -2.1181,E1 24.8494,E2 290.0652} C_DIS
LIN {X -88.3016,Y 28.5004,Z 91,A 157.6762,B 24.9172,C -2.1008,E1 24.8471,E2 287.4311} C_DIS
LIN {X -89.3013,Y 25.1939,Z 91,A 159.8649,B 24.9176,C -2.0958,E1 24.8454,E2 285.2415} C_DIS
LIN {X -90.2504,Y 21.547,Z 91,A 162.2071,B 24.9182,C -2.089,E1 24.8438,E2 282.902} C_DIS
LIN {X -91.0421,Y 17.9143,Z 91,A 164.5026,B 24.9187,C -2.0817,E1 24.8425,E2 280.6105} C_DIS
LIN {X -91.6677,Y 14.3704,Z 91,A 166.6704,B 24.9194,C -2.0729,E1 24.8415,E2 278.4506} C_DIS
LIN {X -92.1392,Y 10.9469,Z 91,A 168.8903,B 24.9197,C -2.0687,E1 24.8407,E2 276.2275} C_DIS
LIN {X -92.5243,Y 6.9885,Z 91,A 171.428,B 24.9202,C -2.0633,E1 24.8401,E2 273.6874} C_DIS
LIN {X -92.7357,Y 3.0964,Z 91,A 173.8005,B 24.9208,C -2.0546,E1 24.8398,E2 271.3216} C_DIS
LIN {X -92.7847,Y -0.6312,Z 91,A 176.101,B 24.9214,C -2.0472,E1 24.8398,E2 269.0249} C_DIS
LIN {X -92.7007,Y -4.0018,Z 91,A 178.111,B 24.9221,C -2.0383,E1 24.84,E2 267.0239} C_DIS
LIN {X -92.4866,Y -7.4612,Z 91,A -179.6546,B 24.9224,C -2.0344,E1 24.8404,E2 264.7854} C_DIS
LIN {X -92.1227,Y -11.0861,Z 91,A -177.3763,B 24.9229,C -2.0282,E1 24.8411,E2 262.5083} C_DIS
LIN {X -91.6453,Y -14.5153,Z 91,A -175.1904,B 24.9233,C -2.0229,E1 24.842,E2 260.3219} C_DIS
LIN {X -90.9759,Y -18.2447,Z 91,A -172.8943,B 24.9239,C -2.0143,E1 24.8432,E2 258.0328} C_DIS
LIN {X -90.2022,Y -21.7488,Z 91,A -170.5831,B 24.9242,C -2.0105,E1 24.8447,E2 255.7172} C_DIS
LIN {X -89.4245,Y -24.7538,Z 91,A -167.8605,B 24.9227,C -2.0299,E1 24.8468,E2 252.9325} C_DIS
LIN {X -88.0339,Y -29.3173,Z 91,A -165.7782,B 24.9254,C -1.994,E1 24.8485,E2 250.9238} C_DIS
LIN {X -86.2056,Y -34.3222,Z 91,A -162.5149,B 24.9262,C -1.9835,E1 24.8517,E2 247.6671} C_DIS
LIN {X -84.8914,Y -37.4555,Z 91,A -160.351,B 24.9265,C -1.9796,E1 24.8541,E2 245.5007} C_DIS
LIN {X -83.8986,Y -39.6292,Z 91,A -158.5734,B 24.9261,C -1.9849,E1 24.8563,E2 243.7007} C_DIS
LIN {X -81.8385,Y -43.7273,Z 91,A -155.9772,B 24.9273,C -1.9697,E1 24.8596,E2 241.127} C_DIS
LIN {X -80.0925,Y -46.8488,Z 91,A -154.0443,B 24.9283,C -1.9552,E1 24.8622,E2 239.2187} C_DIS
LIN {X -78.488,Y -49.4897,Z 91,A -151.8059,B 24.9279,C -1.9606,E1 24.8655,E2 236.9559} C_DIS
LIN {X -76.6448,Y -52.2983,Z 91,A -149.5853,B 24.9279,C -1.96,E1 24.869,E2 234.7257} C_DIS
LIN {X -74.2002,Y -55.7115,Z 91,A -147.2341,B 24.929,C -1.9459,E1 24.8728,E2 232.3966} C_DIS
LIN {X -72.1108,Y -58.3906,Z 91,A -145.1022,B 24.9293,C -1.942,E1 24.8765,E2 230.2639} C_DIS
LIN {X -69.4471,Y -61.5362,Z 91,A -142.4778,B 24.9295,C -1.9387,E1 24.8813,E2 227.6354} C_DIS
LIN {X -67.0363,Y -64.1536,Z 91,A -140.2914,B 24.9299,C -1.9336,E1 24.8855,E2 225.4517} C_DIS
LIN {X -65.1722,Y -66.0457,Z 91,A -138.5984,B 24.93,C -1.9319,E1 24.8889,E2 223.7557} C_DIS
LIN {X -62.4004,Y -68.6719,Z 91,A -136.239,B 24.9304,C -1.9271,E1 24.8937,E2 221.398} C_DIS
LIN {X -59.7526,Y -70.9874,Z 91,A -134.0498,B 24.9306,C -1.9236,E1 24.8984,E2 219.2088} C_DIS
LIN {X -56.7817,Y -73.3847,Z 91,A -131.7603,B 24.9311,C -1.9171,E1 24.9034,E2 216.9262} C_DIS
LIN {X -53.489,Y -75.8194,Z 91,A -129.1879,B 24.9313,C -1.9142,E1 24.9092,E2 214.3517} C_DIS
LIN {X -50.7053,Y -77.708,Z 91,A -127.0937,B 24.9315,C -1.9115,E1 24.914,E2 212.2571} C_DIS
LIN {X -47.7199,Y -79.5768,Z 91,A -124.9019,B 24.9317,C -1.9088,E1 24.9193,E2 210.0648} C_DIS
LIN {X -44.9322,Y -81.1828,Z 91,A -123.1311,B 24.9324,C -1.899,E1 24.9235,E2 208.3122} C_DIS
LIN {X -42.3071,Y -82.5806,Z 91,A -121.3321,B 24.9327,C -1.8954,E1 24.928,E2 206.5168} C_DIS
LIN {X -39.4757,Y -83.9716,Z 91,A -119.1046,B 24.9322,C -1.9023,E1 24.9336,E2 204.267} C_DIS
LIN {X -36.2543,Y -85.4115,Z 91,A -116.9727,B 24.9324,C -1.8984,E1 24.9391,E2 202.1394} C_DIS
LIN {X -33.1086,Y -86.6793,Z 91,A -114.9039,B 24.9326,C -1.8956,E1 24.9444,E2 200.0729} C_DIS
LIN {X -30.306,Y -87.6991,Z 91,A -112.9867,B 24.9326,C -1.8965,E1 24.9495,E2 198.1497} C_DIS
LIN {X -27.217,Y -88.706,Z 91,A -111.098,B 24.933,C -1.8911,E1 24.9545,E2 196.2706} C_DIS
LIN {X -22.6743,Y -89.9743,Z 91,A -107.5532,B 24.9316,C -1.9108,E1 24.9642,E2 192.6737} C_DIS
LIN {X -19.149,Y -90.79,Z 91,A -105.815,B 24.9328,C -1.8928,E1 24.9689,E2 190.976} C_DIS
LIN {X -14.7111,Y -91.6132,Z 91,A -103.0152,B 24.9328,C -1.8924,E1 24.9766,E2 188.1745} C_DIS
LIN {X -10.6555,Y -92.1725,Z 91,A -100.2115,B 24.9322,C -1.9014,E1 24.9844,E2 185.3473} C_DIS
LIN {X -7.3382,Y -92.4964,Z 91,A -98.0643,B 24.932,C -1.9044,E1 24.9904,E2 183.1921} C_DIS
LIN {X -1.871,Y -92.7683,Z 91,A -94.8232,B 24.9323,C -1.9,E1 24.9994,E2 179.961} C_DIS
Enddeposition()
END
